FUNCTION "dos_comp_7" : VOID	// FC 9
TITLE = Dosing component 7
VERSION : 0.1
VAR_TEMP
  dosi_man : BOOL ;
END_VAR
BEGIN
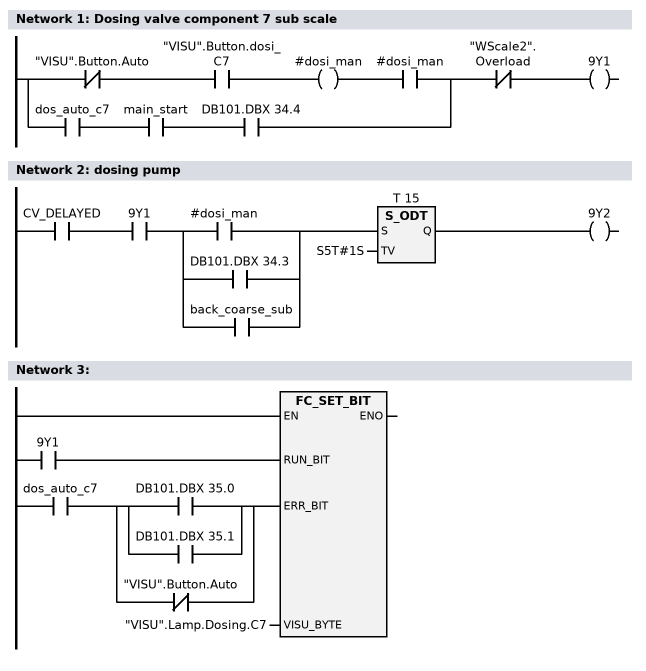
NETWORK
TITLE = Dosing valve component 7 sub scale
//automatic and manual steps
      A(;
      AN    "VISU".Button.Auto;
      A     "VISU".Button.dosi_C7;
      =     #dosi_man;
      A     #dosi_man;
      O;
      A     "dos_auto_c7";
      A     "main_start";
      A     DB101.DBX 34.4;
      );
      AN    "WScale2".Overload;
      =     "9Y1";
NETWORK
TITLE = dosing pump
//automatic and manual steps
      A     "CV_DELAYED";
      A     "9Y1";
      A(;
      O     #dosi_man;
      O     DB101.DBX 34.3;
      O     "back_coarse_sub";
      );
      L     S5T#1S;
      SD    T 15;
      NOP   0;
      NOP   0;
      NOP   0;
      A     T 15;
      =     "9Y2";
NETWORK
TITLE =
      A     "9Y1";
      =     L 1.0;
      BLD   103;
      A     "dos_auto_c7";
      A(;
      O     DB101.DBX 35.0;
      O     DB101.DBX 35.1;
      ON    "VISU".Button.Auto;
      );
      =     L 1.1;
      BLD   103;
      CALL  "FC_SET_BIT" (
           RUN_BIT                  := L 1.0,
           ERR_BIT                  := L 1.1,
           VISU_BYTE                := "VISU".Lamp.Dosing.C7);
      NOP   0;
END_FUNCTION

FUNCTION "dos_comp_8" : VOID	// FC 10
TITLE = Dosing component 8
VERSION : 0.1
VAR_TEMP
  dosi_man : BOOL ;
END_VAR
BEGIN
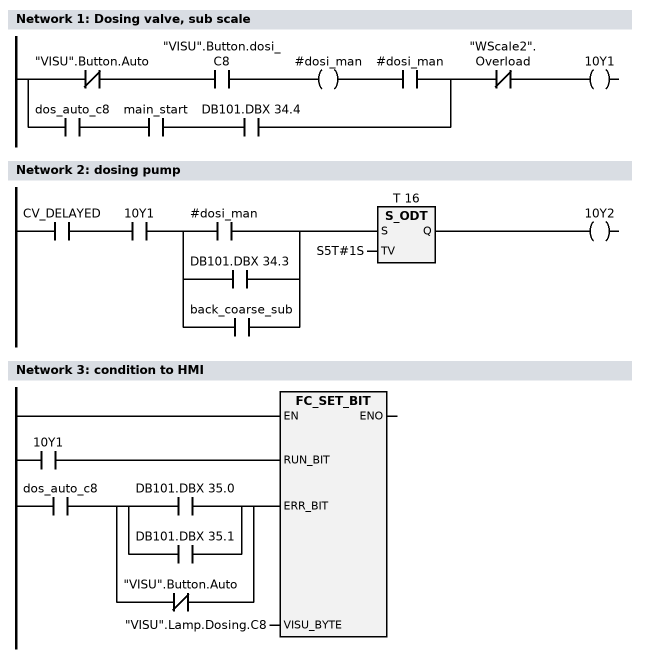
NETWORK
TITLE = Dosing valve, sub scale
//automatic and manual steps
      A(;
      AN    "VISU".Button.Auto;
      A     "VISU".Button.dosi_C8;
      =     #dosi_man;
      A     #dosi_man;
      O;
      A     "dos_auto_c8";
      A     "main_start";
      A     DB101.DBX 34.4;
      );
      AN    "WScale2".Overload;
      =     "10Y1";
NETWORK
TITLE = dosing pump
//automatic and manual steps
      A     "CV_DELAYED";
      A     "10Y1";
      A(;
      O     #dosi_man;
      O     DB101.DBX 34.3;
      O     "back_coarse_sub";
      );
      L     S5T#1S;
      SD    T 16;
      NOP   0;
      NOP   0;
      NOP   0;
      A     T 16;
      =     "10Y2";
NETWORK
TITLE = condition to HMI 
      A     "10Y1";
      =     L 1.0;
      BLD   103;
      A     "dos_auto_c8";
      A(;
      O     DB101.DBX 35.0;
      O     DB101.DBX 35.1;
      ON    "VISU".Button.Auto;
      );
      =     L 1.1;
      BLD   103;
      CALL  "FC_SET_BIT" (
           RUN_BIT                  := L 1.0,
           ERR_BIT                  := L 1.1,
           VISU_BYTE                := "VISU".Lamp.Dosing.C8);
      NOP   0;
END_FUNCTION

FUNCTION "dos_comp_9" : VOID	// FC 11
TITLE = Dosing component 9
VERSION : 0.1
VAR_TEMP
  dosi_man : BOOL ;
END_VAR
BEGIN
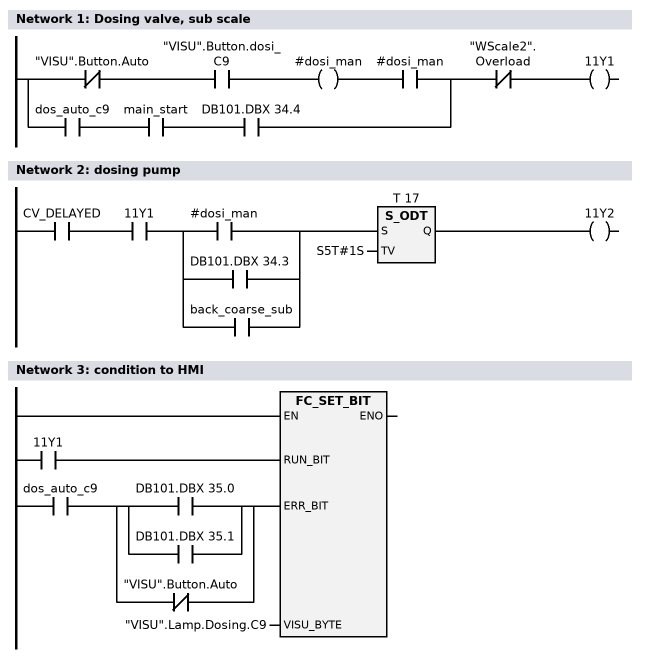
NETWORK
TITLE = Dosing valve, sub scale
//automatic and manual steps
      A(;
      AN    "VISU".Button.Auto;
      A     "VISU".Button.dosi_C9;
      =     #dosi_man;
      A     #dosi_man;
      O;
      A     "dos_auto_c9";
      A     "main_start";
      A     DB101.DBX 34.4;
      );
      AN    "WScale2".Overload;
      =     "11Y1";
NETWORK
TITLE = dosing pump
//automatic and manual steps
      A     "CV_DELAYED";
      A     "11Y1";
      A(;
      O     #dosi_man;
      O     DB101.DBX 34.3;
      O     "back_coarse_sub";
      );
      L     S5T#1S;
      SD    T 17;
      NOP   0;
      NOP   0;
      NOP   0;
      A     T 17;
      =     "11Y2";
NETWORK
TITLE = condition to HMI 
      A     "11Y1";
      =     L 1.0;
      BLD   103;
      A     "dos_auto_c9";
      A(;
      O     DB101.DBX 35.0;
      O     DB101.DBX 35.1;
      ON    "VISU".Button.Auto;
      );
      =     L 1.1;
      BLD   103;
      CALL  "FC_SET_BIT" (
           RUN_BIT                  := L 1.0,
           ERR_BIT                  := L 1.1,
           VISU_BYTE                := "VISU".Lamp.Dosing.C9);
      NOP   0;
END_FUNCTION

FUNCTION "dos_comp_10" : VOID	// FC 12
TITLE = Dosing component 10
VERSION : 0.1
VAR_TEMP
  dosi_man : BOOL ;
END_VAR
BEGIN
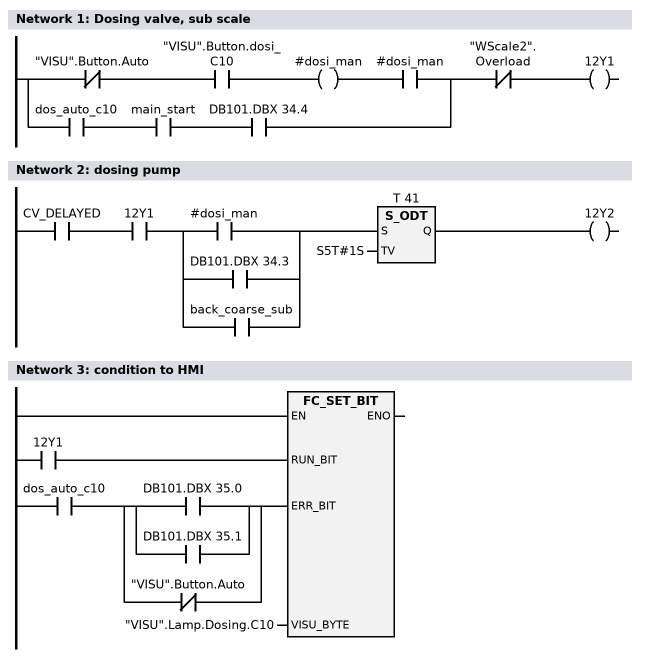
NETWORK
TITLE = Dosing valve, sub scale
//automatic and manual steps
      A(;
      AN    "VISU".Button.Auto;
      A     "VISU".Button.dosi_C10;
      =     #dosi_man;
      A     #dosi_man;
      O;
      A     "dos_auto_c10";
      A     "main_start";
      A     DB101.DBX 34.4;
      );
      AN    "WScale2".Overload;
      =     "12Y1";
NETWORK
TITLE = dosing pump
//automatic and manual steps
      A     "CV_DELAYED";
      A     "12Y1";
      A(;
      O     #dosi_man;
      O     DB101.DBX 34.3;
      O     "back_coarse_sub";
      );
      L     S5T#1S;
      SD    T 41;
      NOP   0;
      NOP   0;
      NOP   0;
      A     T 41;
      =     "12Y2";
NETWORK
TITLE = condition to HMI
      A     "12Y1";
      =     L 1.0;
      BLD   103;
      A     "dos_auto_c10";
      A(;
      O     DB101.DBX 35.0;
      O     DB101.DBX 35.1;
      ON    "VISU".Button.Auto;
      );
      =     L 1.1;
      BLD   103;
      CALL  "FC_SET_BIT" (
           RUN_BIT                  := L 1.0,
           ERR_BIT                  := L 1.1,
           VISU_BYTE                := "VISU".Lamp.Dosing.C10);
      NOP   0;
END_FUNCTION

FUNCTION "dos_comp_11" : VOID	// FC 13
TITLE = Dosing component 11
VERSION : 0.1
VAR_TEMP
  dosi_man : BOOL ;
END_VAR
BEGIN
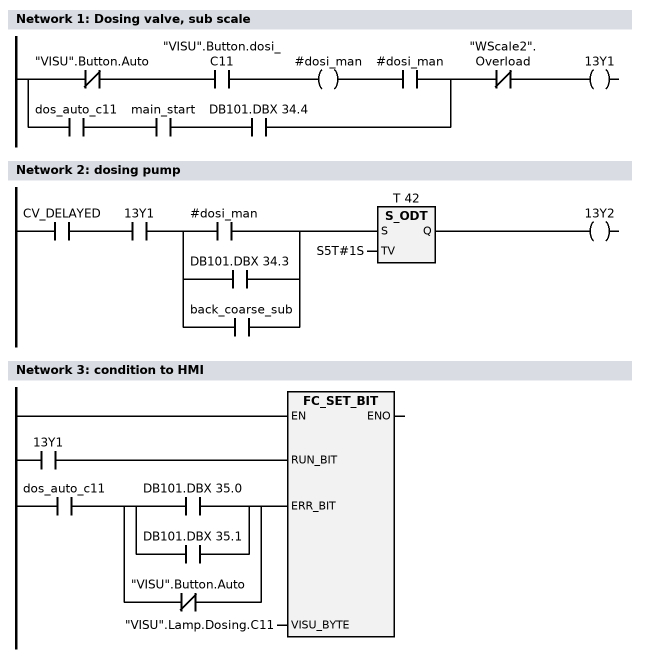
NETWORK
TITLE = Dosing valve, sub scale
//automatic and manual steps
      A(;
      AN    "VISU".Button.Auto;
      A     "VISU".Button.dosi_C11;
      =     #dosi_man;
      A     #dosi_man;
      O;
      A     "dos_auto_c11";
      A     "main_start";
      A     DB101.DBX 34.4;
      );
      AN    "WScale2".Overload;
      =     "13Y1";
NETWORK
TITLE = dosing pump
//automatic and manual steps
      A     "CV_DELAYED";
      A     "13Y1";
      A(;
      O     #dosi_man;
      O     DB101.DBX 34.3;
      O     "back_coarse_sub";
      );
      L     S5T#1S;
      SD    T 42;
      NOP   0;
      NOP   0;
      NOP   0;
      A     T 42;
      =     "13Y2";
NETWORK
TITLE = condition to HMI
      A     "13Y1";
      =     L 1.0;
      BLD   103;
      A     "dos_auto_c11";
      A(;
      O     DB101.DBX 35.0;
      O     DB101.DBX 35.1;
      ON    "VISU".Button.Auto;
      );
      =     L 1.1;
      BLD   103;
      CALL  "FC_SET_BIT" (
           RUN_BIT                  := L 1.0,
           ERR_BIT                  := L 1.1,
           VISU_BYTE                := "VISU".Lamp.Dosing.C11);
      NOP   0;
END_FUNCTION

FUNCTION "dos_comp_12" : VOID	// FC 14
TITLE = Dosing component 12
VERSION : 0.1
VAR_TEMP
  dosi_man : BOOL ;
END_VAR
BEGIN
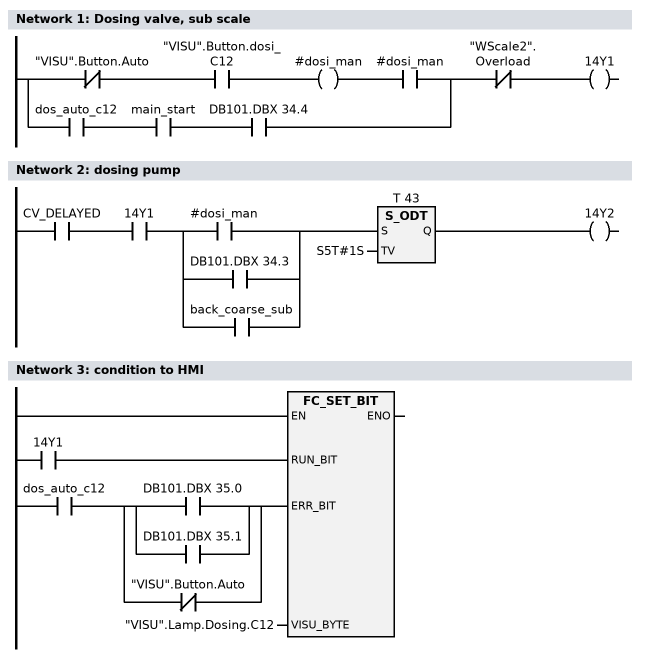
NETWORK
TITLE = Dosing valve, sub scale
//automatic and manual steps
      A(;
      AN    "VISU".Button.Auto;
      A     "VISU".Button.dosi_C12;
      =     #dosi_man;
      A     #dosi_man;
      O;
      A     "dos_auto_c12";
      A     "main_start";
      A     DB101.DBX 34.4;
      );
      AN    "WScale2".Overload;
      =     "14Y1";
NETWORK
TITLE = dosing pump
//automatic and manual steps
      A     "CV_DELAYED";
      A     "14Y1";
      A(;
      O     #dosi_man;
      O     DB101.DBX 34.3;
      O     "back_coarse_sub";
      );
      L     S5T#1S;
      SD    T 43;
      NOP   0;
      NOP   0;
      NOP   0;
      A     T 43;
      =     "14Y2";
NETWORK
TITLE = condition to HMI
      A     "14Y1";
      =     L 1.0;
      BLD   103;
      A     "dos_auto_c12";
      A(;
      O     DB101.DBX 35.0;
      O     DB101.DBX 35.1;
      ON    "VISU".Button.Auto;
      );
      =     L 1.1;
      BLD   103;
      CALL  "FC_SET_BIT" (
           RUN_BIT                  := L 1.0,
           ERR_BIT                  := L 1.1,
           VISU_BYTE                := "VISU".Lamp.Dosing.C12);
      NOP   0;
END_FUNCTION

FUNCTION "discharge_main_scale" : VOID	// FC 22
TITLE = discharge mainscale
VERSION : 0.0
VAR_TEMP
  disc_auto : BOOL ;
  disc1 : BOOL ;
  disc2 : BOOL ;
  disc3 : BOOL ;
END_VAR
BEGIN
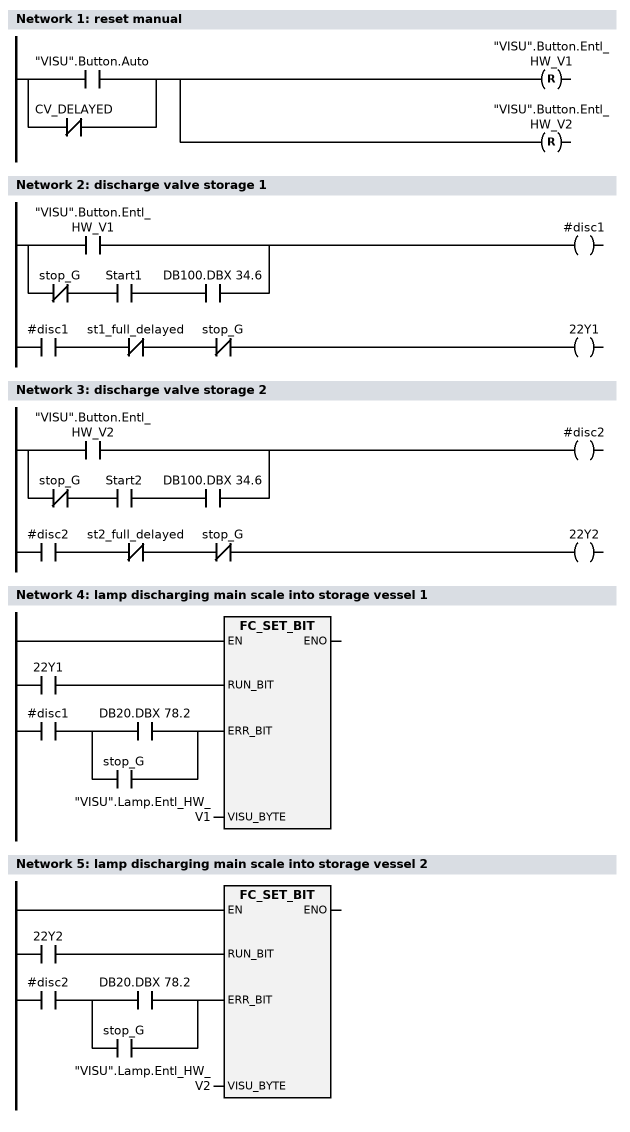
NETWORK
TITLE = reset manual
      O     "VISU".Button.Auto;
      ON    "CV_DELAYED";
      R     "VISU".Button.Entl_HW_V1;
      R     "VISU".Button.Entl_HW_V2;
NETWORK
TITLE = discharge valve storage 1
      A(;
      O     "VISU".Button.Entl_HW_V1;
      O;
      AN    "stop_G";
      A     "Start1";
      A     DB100.DBX 34.6;
      );
      =     #disc1;
      A     #disc1;
      AN    "st1_full_delayed";
      AN    "stop_G";
      =     "22Y1";
NETWORK
TITLE = discharge valve storage 2
      A(;
      O     "VISU".Button.Entl_HW_V2;
      O;
      AN    "stop_G";
      A     "Start2";
      A     DB100.DBX 34.6;
      );
      =     #disc2;
      A     #disc2;
      AN    "st2_full_delayed";
      AN    "stop_G";
      =     "22Y2";
NETWORK
TITLE = lamp discharging main scale into storage vessel 1
      A     "22Y1";
      =     L 1.0;
      BLD   103;
      A     #disc1;
      A(;
      O     DB20.DBX 78.2;
      O     "stop_G";
      );
      =     L 1.1;
      BLD   103;
      CALL  "FC_SET_BIT" (
           RUN_BIT                  := L 1.0,
           ERR_BIT                  := L 1.1,
           VISU_BYTE                := "VISU".Lamp.Entl_HW_V1);
      NOP   0;
NETWORK
TITLE = lamp discharging main scale into storage vessel 2
      A     "22Y2";
      =     L 1.0;
      BLD   103;
      A     #disc2;
      A(;
      O     DB20.DBX 78.2;
      O     "stop_G";
      );
      =     L 1.1;
      BLD   103;
      CALL  "FC_SET_BIT" (
           RUN_BIT                  := L 1.0,
           ERR_BIT                  := L 1.1,
           VISU_BYTE                := "VISU".Lamp.Entl_HW_V2);
      NOP   0;
END_FUNCTION

FUNCTION "discharge_sub_scale" : VOID	// FC 23
TITLE = discharge  sub scale
VERSION : 0.1
VAR_TEMP
  disc : BOOL ;
END_VAR
BEGIN
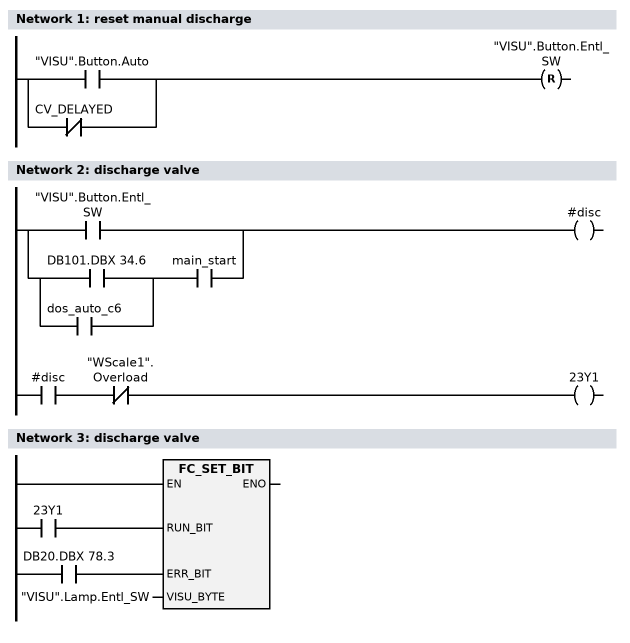
NETWORK
TITLE = reset manual discharge
      O     "VISU".Button.Auto;
      ON    "CV_DELAYED";
      R     "VISU".Button.Entl_SW;
NETWORK
TITLE = discharge valve
      A(;
      O     "VISU".Button.Entl_SW;
      O;
      A(;
      O     DB101.DBX 34.6;
      O     "dos_auto_c6";
      );
      A     "main_start";
      );
      =     #disc;
      A     #disc;
      AN    "WScale1".Overload;
      =     "23Y1";
NETWORK
TITLE = discharge valve
      A     "23Y1";
      =     L 1.0;
      BLD   103;
      A     DB20.DBX 78.3;
      =     L 1.1;
      BLD   103;
      CALL  "FC_SET_BIT" (
           RUN_BIT                  := L 1.0,
           ERR_BIT                  := L 1.1,
           VISU_BYTE                := "VISU".Lamp.Entl_SW);
      NOP   0;
END_FUNCTION

FUNCTION "agit_MS" : VOID	// FC 25
TITLE = main scale, agitator
VERSION : 0.1
BEGIN
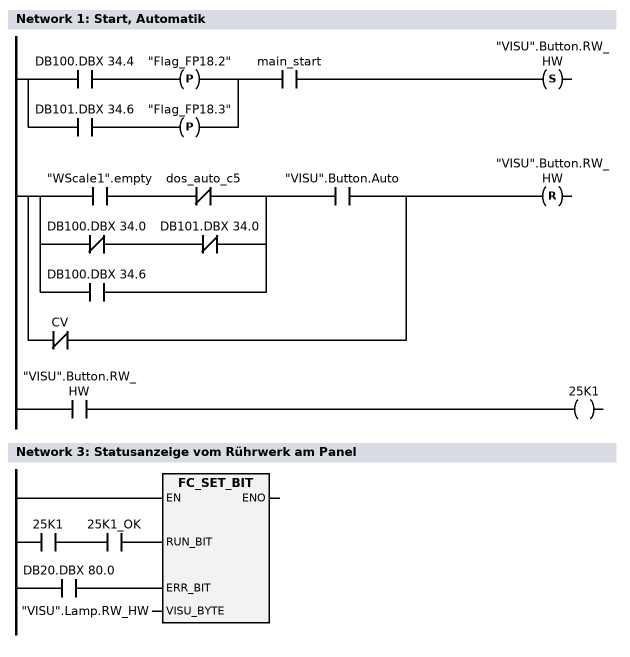
NETWORK
TITLE = Start, Automatik
      A(;
      A     DB100.DBX 34.4;
      FP    "Flag_FP18.2";
      O(;
      A     DB101.DBX 34.6;
      FP    "Flag_FP18.3";
      );
      );
      A     "main_start";
      S     "VISU".Button.RW_HW;
      A(;
      A(;
      A     "WScale1".empty;
      AN    "dos_auto_c5";
      O;
      AN    DB100.DBX 34.0;
      AN    DB101.DBX 34.0;
      O     DB100.DBX 34.6;
      );
      A     "VISU".Button.Auto;
      ON    "CV";
      );
      R     "VISU".Button.RW_HW;
      A     "VISU".Button.RW_HW;
      =     "25K1";
NETWORK
TITLE = Schütz auf Rückmeldung prüfen
      A(;
      X     "25K1";
      X     "25K1_OK";
      );
      A     "CV_DELAYED";
      L     S5T#1S;
      SD    T 18;
      NOP   0;
      NOP   0;
      NOP   0;
      A     T 18;
      =     DB20.DBX 80.0;
NETWORK
TITLE = Statusanzeige vom Rührwerk am Panel
      A     "25K1";
      A     "25K1_OK";
      =     L 0.0;
      BLD   103;
      A     DB20.DBX 80.0;
      =     L 0.1;
      BLD   103;
      CALL  "FC_SET_BIT" (
           RUN_BIT                  := L 0.0,
           ERR_BIT                  := L 0.1,
           VISU_BYTE                := "VISU".Lamp.RW_HW);
      NOP   0;
END_FUNCTION

FUNCTION "aigt_level_storage1" : VOID	// FC 26
TITLE = agit_level storage vessel 1
VERSION : 0.1
VAR_TEMP
  imp : BOOL ;
END_VAR
BEGIN
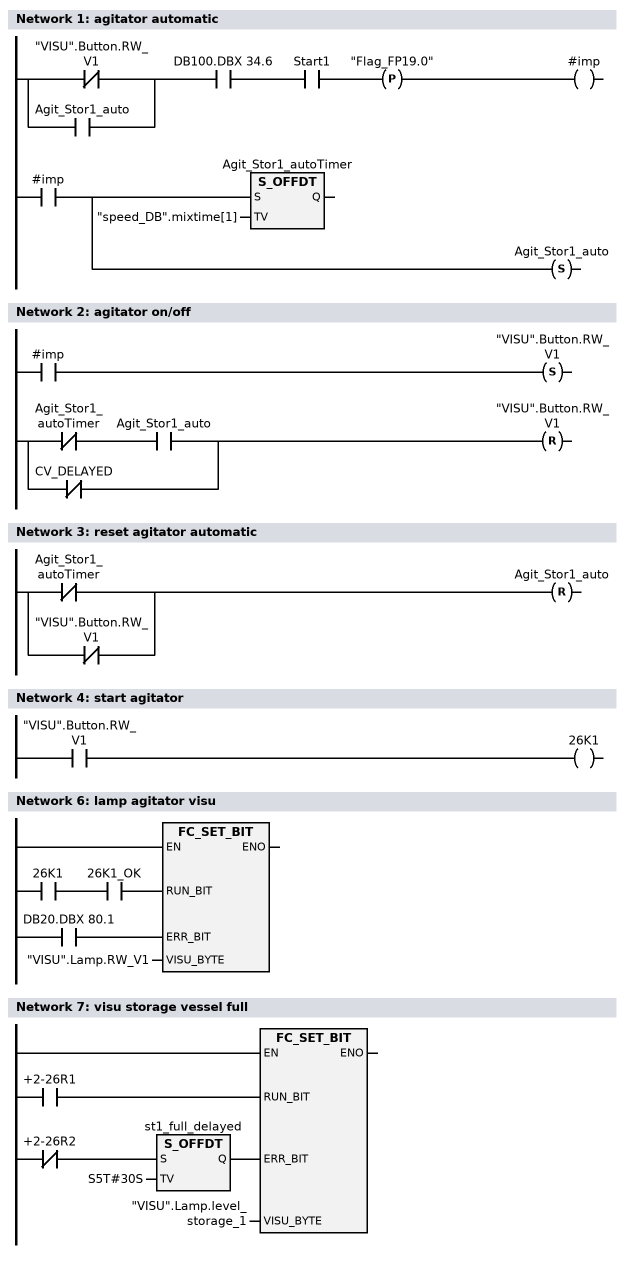
NETWORK
TITLE = agitator automatic
      A(;
      ON    "VISU".Button.RW_V1;
      O     "Agit_Stor1_auto";
      );
      A     DB100.DBX 34.6;
      A     "Start1";
      FP    "Flag_FP19.0";
      =     #imp;
      A     #imp;
      =     L 1.0;
      A     L 1.0;
      L     "speed_DB".mixtime[1];
      SF    "Agit_Stor1_autoTimer";
      NOP   0;
      NOP   0;
      NOP   0;
      NOP   0;
      A     L 1.0;
      BLD   102;
      S     "Agit_Stor1_auto";
NETWORK
TITLE = agitator on/off
      A     #imp;
      S     "VISU".Button.RW_V1;
      A(;
      AN    "Agit_Stor1_autoTimer";
      A     "Agit_Stor1_auto";
      ON    "CV_DELAYED";
      );
      R     "VISU".Button.RW_V1;
      NOP   0;
NETWORK
TITLE = reset agitator automatic
      ON    "Agit_Stor1_autoTimer";
      ON    "VISU".Button.RW_V1;
      R     "Agit_Stor1_auto";
NETWORK
TITLE = start agitator
      A     "VISU".Button.RW_V1;
      =     "26K1";
NETWORK
TITLE = fault contactor/circuit breaker
      A(;
      X     "26K1";
      X     "26K1_OK";
      );
      A     "CV_DELAYED";
      L     S5T#1S;
      SD    T 10;
      NOP   0;
      NOP   0;
      NOP   0;
      A     T 10;
      =     DB20.DBX 80.1;
NETWORK
TITLE = lamp agitator visu
      A     "26K1";
      A     "26K1_OK";
      =     L 1.0;
      BLD   103;
      A     DB20.DBX 80.1;
      =     L 1.1;
      BLD   103;
      CALL  "FC_SET_BIT" (
           RUN_BIT                  := L 1.0,
           ERR_BIT                  := L 1.1,
           VISU_BYTE                := "VISU".Lamp.RW_V1);
      NOP   0;
NETWORK
TITLE = visu storage vessel full
      A     "+2-26R1";
      =     L 1.0;
      BLD   103;
      A(;
      AN    "+2-26R2";
      L     S5T#30S;
      SF    "st1_full_delayed";
      NOP   0;
      NOP   0;
      NOP   0;
      A     "st1_full_delayed";
      );
      =     L 1.1;
      BLD   103;
      CALL  "FC_SET_BIT" (
           RUN_BIT                  := L 1.0,
           ERR_BIT                  := L 1.1,
           VISU_BYTE                := "VISU".Lamp.level_storage_1);
      NOP   0;
END_FUNCTION

FUNCTION "aigt_level_storage2" : VOID	// FC 27
TITLE = agit_level storage vessel 2
VERSION : 0.1
VAR_TEMP
  imp : BOOL ;
END_VAR
BEGIN
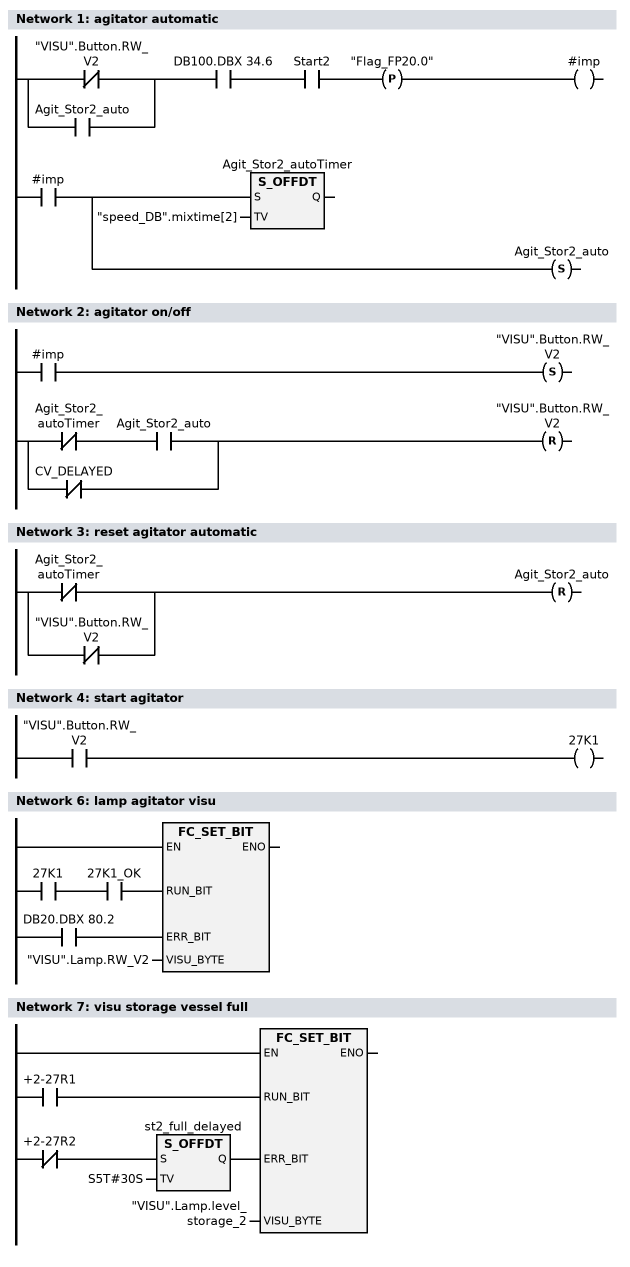
NETWORK
TITLE = agitator automatic
      A(;
      ON    "VISU".Button.RW_V2;
      O     "Agit_Stor2_auto";
      );
      A     DB100.DBX 34.6;
      A     "Start2";
      FP    "Flag_FP20.0";
      =     #imp;
      A     #imp;
      =     L 1.0;
      A     L 1.0;
      L     "speed_DB".mixtime[2];
      SF    "Agit_Stor2_autoTimer";
      NOP   0;
      NOP   0;
      NOP   0;
      NOP   0;
      A     L 1.0;
      BLD   102;
      S     "Agit_Stor2_auto";
NETWORK
TITLE = agitator on/off
      A     #imp;
      S     "VISU".Button.RW_V2;
      A(;
      AN    "Agit_Stor2_autoTimer";
      A     "Agit_Stor2_auto";
      ON    "CV_DELAYED";
      );
      R     "VISU".Button.RW_V2;
      NOP   0;
NETWORK
TITLE = reset agitator automatic
      ON    "Agit_Stor2_autoTimer";
      ON    "VISU".Button.RW_V2;
      R     "Agit_Stor2_auto";
NETWORK
TITLE = start agitator
      A     "VISU".Button.RW_V2;
      =     "27K1";
NETWORK
TITLE = fault contactor/circuit breaker
      A(;
      X     "27K1";
      X     "27K1_OK";
      );
      A     "CV_DELAYED";
      L     S5T#1S;
      SD    T 22;
      NOP   0;
      NOP   0;
      NOP   0;
      A     T 22;
      =     DB20.DBX 80.2;
NETWORK
TITLE = lamp agitator visu
      A     "27K1";
      A     "27K1_OK";
      =     L 1.0;
      BLD   103;
      A     DB20.DBX 80.2;
      =     L 1.1;
      BLD   103;
      CALL  "FC_SET_BIT" (
           RUN_BIT                  := L 1.0,
           ERR_BIT                  := L 1.1,
           VISU_BYTE                := "VISU".Lamp.RW_V2);
      NOP   0;
NETWORK
TITLE = visu storage vessel full
      A     "+2-27R1";
      =     L 1.0;
      BLD   103;
      A(;
      AN    "+2-27R2";
      L     S5T#30S;
      SF    "st2_full_delayed";
      NOP   0;
      NOP   0;
      NOP   0;
      A     "st2_full_delayed";
      );
      =     L 1.1;
      BLD   103;
      CALL  "FC_SET_BIT" (
           RUN_BIT                  := L 1.0,
           ERR_BIT                  := L 1.1,
           VISU_BYTE                := "VISU".Lamp.level_storage_2);
      NOP   0;
END_FUNCTION

FUNCTION "filling_vat" : VOID	// FC 29
TITLE = Vat VITS filling out from storage 1
VERSION : 0.1
VAR_TEMP
  valve_1 : BOOL ;
  valve_2 : BOOL ;
END_VAR
BEGIN
NETWORK
TITLE = Filling ON/OFF
//"VISU".Button.filling_1
      A(;
      A(;
      A     "VISU".Button.filling_1;
      AN    "+4-29R1";
      S     "VITS1_FILLING_ON/OFF";
      A(;
      ON    "VISU".Button.filling_1;
      ON    "+4-29R2";
      );
      R     "VITS1_FILLING_ON/OFF";
      A     "VITS1_FILLING_ON/OFF";
      );
      AN    DB20.DBX 83.0;
      O(;
      A     "VISU".Button.fillvalve_1;
      L     S5T#3S;
      SD    "VITS1_TIPP_TIMER";
      A     "VISU".Button.filling_3;
      R     "VITS1_TIPP_TIMER";
      NOP   0;
      NOP   0;
      A     "VITS1_TIPP_TIMER";
      );
      );
      =     #valve_1;
      A     #valve_1;
      A     "+VTITS-K1";
      L     S5T#1S;
      SF    T 44;
      NOP   0;
      NOP   0;
      NOP   0;
      A     T 44;
      =     "+4-29Y1";
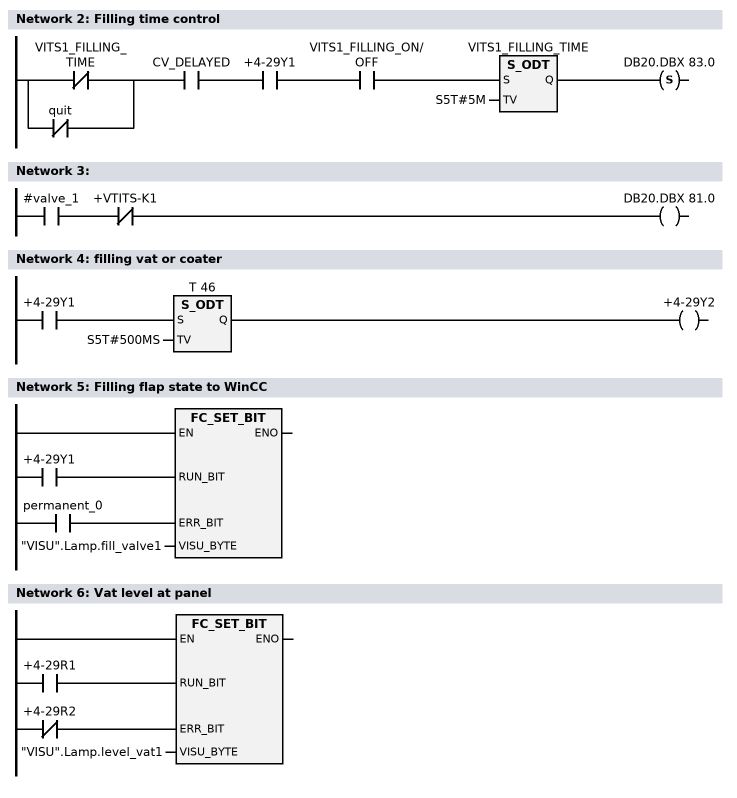
NETWORK
TITLE = Filling time control
      A(;
      ON    "VITS1_FILLING_TIME";
      ON    "quit";
      );
      A     "CV_DELAYED";
      A     "+4-29Y1";
      A     "VITS1_FILLING_ON/OFF";
      L     S5T#5M;
      SD    "VITS1_FILLING_TIME";
      NOP   0;
      NOP   0;
      NOP   0;
      A     "VITS1_FILLING_TIME";
      S     DB20.DBX 83.0;
NETWORK
TITLE =
      A     #valve_1;
      AN    "+VTITS-K1";
      =     DB20.DBX 81.0;
NETWORK
TITLE = filling vat or coater
      A     "+4-29Y1";
      L     S5T#500MS;
      SD    T 46;
      NOP   0;
      NOP   0;
      NOP   0;
      A     T 46;
      =     "+4-29Y2";
NETWORK
TITLE = Filling flap state to WinCC
      A     "+4-29Y1";
      =     L 1.0;
      BLD   103;
      A     "permanent_0";
      =     L 1.1;
      BLD   103;
      CALL  "FC_SET_BIT" (
           RUN_BIT                  := L 1.0,
           ERR_BIT                  := L 1.1,
           VISU_BYTE                := "VISU".Lamp.fill_valve1);
      NOP   0;
NETWORK
TITLE = Vat level at panel
      A     "+4-29R1";
      =     L 1.0;
      BLD   103;
      AN    "+4-29R2";
      =     L 1.1;
      BLD   103;
      CALL  "FC_SET_BIT" (
           RUN_BIT                  := L 1.0,
           ERR_BIT                  := L 1.1,
           VISU_BYTE                := "VISU".Lamp.level_vat1);
      NOP   0;
END_FUNCTION

FUNCTION "filling_coater" : VOID	// FC 30
TITLE = Coater VITS
VERSION : 0.1
BEGIN
NETWORK
TITLE = Filling ON/OFF
//"VISU".Button.filling_2
      A(;
      A     "VISU".Button.filling_2;
      AN    "+4-30R1";
      S     "VITS2_FILLING_ON/OFF";
      A(;
      ON    "VISU".Button.filling_2;
      ON    "+4-30R2";
      );
      R     "VITS2_FILLING_ON/OFF";
      A     "VITS2_FILLING_ON/OFF";
      );
      AN    DB20.DBX 83.1;
      O(;
      A     "VISU".Button.fillvalve_2;
      L     S5T#3S;
      SD    "VITS2_TIPP_TIMER";
      NOP   0;
      NOP   0;
      NOP   0;
      A     "VITS2_TIPP_TIMER";
      );
      =     "+4-30Y1";
      =     "+4-30Y2";
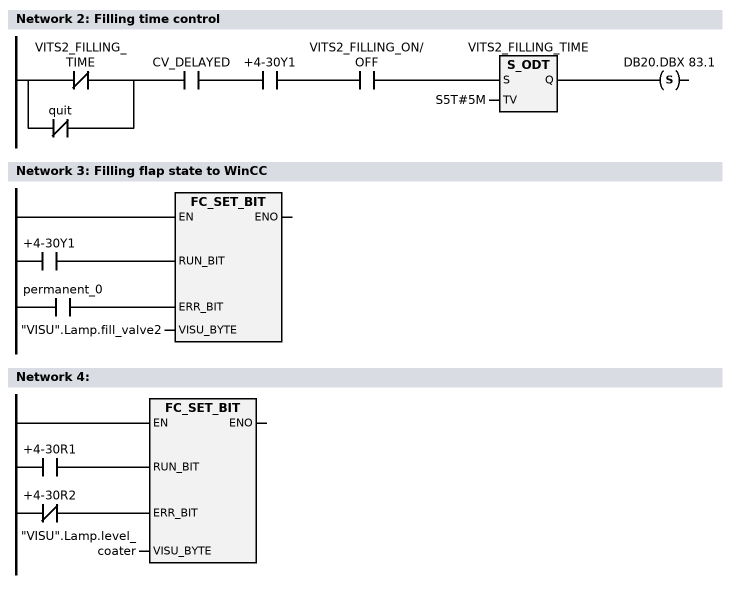
NETWORK
TITLE = Filling time control
      A(;
      ON    "VITS2_FILLING_TIME";
      ON    "quit";
      );
      A     "CV_DELAYED";
      A     "+4-30Y1";
      A     "VITS2_FILLING_ON/OFF";
      L     S5T#5M;
      SD    "VITS2_FILLING_TIME";
      NOP   0;
      NOP   0;
      NOP   0;
      A     "VITS2_FILLING_TIME";
      S     DB20.DBX 83.1;
NETWORK
TITLE = Filling flap state to WinCC
      A     "+4-30Y1";
      =     L 0.0;
      BLD   103;
      A     "permanent_0";
      =     L 0.1;
      BLD   103;
      CALL  "FC_SET_BIT" (
           RUN_BIT                  := L 0.0,
           ERR_BIT                  := L 0.1,
           VISU_BYTE                := "VISU".Lamp.fill_valve2);
      NOP   0;
NETWORK
TITLE =
      A     "+4-30R1";
      =     L 0.0;
      BLD   103;
      AN    "+4-30R2";
      =     L 0.1;
      BLD   103;
      CALL  "FC_SET_BIT" (
           RUN_BIT                  := L 0.0,
           ERR_BIT                  := L 0.1,
           VISU_BYTE                := "VISU".Lamp.level_coater);
      NOP   0;
END_FUNCTION

FUNCTION "coater circ" : VOID	// FC 31
TITLE = Coater circulation
VERSION : 0.1
VAR_TEMP
  fill_time : S5TIME ;
  fill_vat : BOOL ;
END_VAR
BEGIN
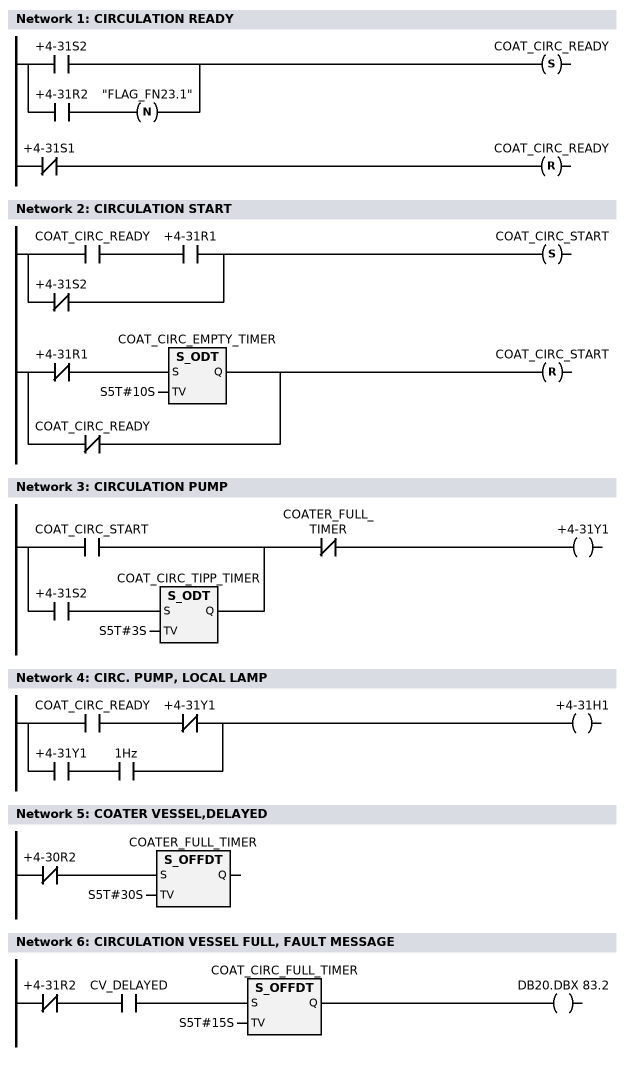
NETWORK
TITLE = CIRCULATION READY
      A(;
      O     "+4-31S2";
      O(;
      A     "+4-31R2";
      FN    "FLAG_FN23.1";
      );
      );
      S     "COAT_CIRC_READY";
      AN    "+4-31S1";
      R     "COAT_CIRC_READY";
      NOP   0;
NETWORK
TITLE = CIRCULATION START
      A(;
      A     "COAT_CIRC_READY";
      A     "+4-31R1";
      ON    "+4-31S2";
      );
      S     "COAT_CIRC_START";
      A(;
      O(;
      AN    "+4-31R1";
      L     S5T#10S;
      SD    "COAT_CIRC_EMPTY_TIMER";
      NOP   0;
      NOP   0;
      NOP   0;
      A     "COAT_CIRC_EMPTY_TIMER";
      );
      ON    "COAT_CIRC_READY";
      );
      R     "COAT_CIRC_START";
      NOP   0;
NETWORK
TITLE = CIRCULATION PUMP
      A(;
      O     "COAT_CIRC_START";
      O(;
      A     "+4-31S2";
      L     S5T#3S;
      SD    "COAT_CIRC_TIPP_TIMER";
      NOP   0;
      NOP   0;
      NOP   0;
      A     "COAT_CIRC_TIPP_TIMER";
      );
      );
      AN    "COATER_FULL_TIMER";
      =     "+4-31Y1";
NETWORK
TITLE = CIRC. PUMP, LOCAL LAMP
      A     "COAT_CIRC_READY";
      AN    "+4-31Y1";
      O;
      A     "+4-31Y1";
      A     "1Hz";
      =     "+4-31H1";
NETWORK
TITLE = COATER VESSEL,DELAYED
      AN    "+4-30R2";
      L     S5T#30S;
      SF    "COATER_FULL_TIMER";
      NOP   0;
      NOP   0;
      NOP   0;
      NOP   0;
NETWORK
TITLE = CIRCULATION VESSEL FULL, FAULT MESSAGE
      AN    "+4-31R2";
      A     "CV_DELAYED";
      L     S5T#15S;
      SF    "COAT_CIRC_FULL_TIMER";
      NOP   0;
      NOP   0;
      NOP   0;
      A     "COAT_CIRC_FULL_TIMER";
      =     DB20.DBX 83.2;
END_FUNCTION

FUNCTION "control_FC" : VOID	// FC 60
TITLE = Control FC
VERSION : 0.1
VAR_TEMP
  t_busy : BOOL ;
END_VAR
BEGIN
NETWORK
TITLE = manual operating
      CALL  "del_ins_line";
      CALL  "Transfer_Recipe";
      CALL  "Rec_handling";
NETWORK
TITLE = zero Gravimet
      L     DB21.DBB 8;	// rem Starts
      L     0;
      <>I;
      AN    "Auto_DB".automatic;
      S     "zero";
      CALL  "zero_FC";
NETWORK
TITLE = scale signals
      A     "cancel_G";
      =     DB100.DBX 34.5;
      =     DB101.DBX 34.5;
      A     "stop_G";
      A     "main_start";
      A     DB100.DBX 34.2;
      =     DB100.DBX 35.5;
      A     "stop_G";
      A     "main_start";
      A     DB101.DBX 34.2;
      =     DB101.DBX 35.5;
      A     "quit";
      R     DB100.DBX 35.2;
      R     DB101.DBX 35.2;
NETWORK
TITLE = Cascading
      L     "Cascad_DW";
      RLD   1;
      T     "Cascad_DW";
NETWORK
TITLE = main scale
      CALL  "SiwarexCS" , "WScale1" (
           ADRESSE                  := 272,
           ABZUGSWAAGE              := FALSE,
           KAS_SIWAREX              := TRUE,
           CPU_Start_Bit            := "CPU_Restart",
           ANLAUFTIMER              := "StartupTimer",
           Quitt                    := "quit",
           StillTimer               := T 100,
           EmptyTimer               := T 101,
           DosiControlTimer         := T 102,
           StepTimer                := T 103);
      CALL  "Dosing" , "DScale1" (
           scale_nr                 := 1,
           Work_DB                  := 26,
           Weigh_DB                 := 10,
           mix_timer                := T 104,
           step_scale1              := "Auto_DB".Step_scale1,
           step_scale2              := "Auto_DB".Step_scale2,
           step_scale3              := "init_DB".max_step,
           step_scale4              := "init_DB".max_step,
           Dosi_Bits                := "Dosibits");
NETWORK
TITLE = Timers
      L     T 101;
      A     "WScale1".discharge;
      JC    M001;
      L     T 103;
      A     "WScale1".StepTime;
      JC    M001;
      L     T 104;
      A     DB100.DBX 35.4;
      JC    M001;
      L     0;
M001: L     60;
      /I;
      T     "HMI_DB".Scale1_timers;
NETWORK
TITLE = fault messages
      A     DB100.DBX 35.0;
      S     DB20.DBX 73.1;
      A     DB100.DBX 35.1;
      AN    DB100.DBX 35.5;
      S     DB20.DBX 73.2;
      A     DB100.DBX 35.5;
      S     DB20.DBX 73.3;
NETWORK
TITLE = sub scale
      CALL  "SiwarexCS" , "WScale2" (
           ADRESSE                  := 280,
           ABZUGSWAAGE              := FALSE,
           KAS_SIWAREX              := TRUE,
           CPU_Start_Bit            := "CPU_Restart",
           ANLAUFTIMER              := "StartupTimer",
           Quitt                    := "quit",
           StillTimer               := T 105,
           EmptyTimer               := T 106,
           DosiControlTimer         := T 107,
           StepTimer                := T 108);
      CALL  "Dosing" , "DScale2" (
           scale_nr                 := 2,
           Work_DB                  := 26,
           Weigh_DB                 := 11,
           mix_timer                := T 109,
           step_scale1              := "Auto_DB".Step_scale1,
           step_scale2              := "Auto_DB".Step_scale2,
           step_scale3              := "init_DB".max_step,
           step_scale4              := "init_DB".max_step,
           Dosi_Bits                := "Dosibits");
NETWORK
TITLE = Timers
      L     T 106;
      A     "WScale2".discharge;
      JC    M002;
      L     T 108;
      A     "WScale2".StepTime;
      JC    M002;
      L     T 109;
      A     DB101.DBX 35.4;
      JC    M002;
      L     0;
M002: L     60;
      /I;
      T     "HMI_DB".Scale2_timers;
NETWORK
TITLE = fault messages sub scale
      A     DB101.DBX 35.0;
      S     DB20.DBX 72.1;
      A     DB101.DBX 35.1;
      AN    DB101.DBX 35.5;
      S     DB20.DBX 72.2;
      A     DB101.DBX 35.5;
      S     DB20.DBX 72.3;
NETWORK
TITLE = rated value total main scale while discharging sub scale
      A     DB101.DBX 34.6;
      FP    "Flag_FP211.0";
      JCN   M003;
      L     DB101.DBD 44;
      L     DB100.DBD 44;
      +R;
      T     DB100.DBD 44;
      L     0;
      T     DB100.DBD 22;
M003: NOP   0;
NETWORK
TITLE = clear starts Gravimet
      AN    "zero";
      AN    DB100.DBX 34.0;
      AN    DB101.DBX 34.0;
      R     "Auto_DB".automatic;
      S     "del_starts_G";
END_FUNCTION

FUNCTION "zero_FC" : VOID	// FC 61
TITLE = Waage nullen
//know_how_protect
//
VERSION : 0.0
VAR_TEMP
  loop_ctr1 : INT ;
  loop_ctr2 : INT ;
  Sum_comp : INT ;
  comp_nr : INT ;
  action : INT ;
  scale_nr : INT ;
  DB_ptr : INT ;
  percent : REAL ;
  Sum_main : REAL ;
  Sum_Sub : REAL ;
  Sum_Col : REAL ;
  Rated_val : REAL ;
  Sum_ptr : DINT ;
  Col_flag : BOOL ;
  Temp_err : BOOL ;
  ptr1 : DINT ;
  ptr2 : DINT ;
  recipe : INT ;
  agit_time : INT ;
  Work_DB : INT ;
  CP_DB : INT ;
  Rec_DB : INT ;
  db_write_CP_date : WORD ;
END_VAR
BEGIN
NETWORK
TITLE = Startnummer bestimmen
      AN    "zero";
      BEC;
      L     0;
      A     "Auto_DB".rem_start1;
      JC    M001;
      L     1;
      A     "Auto_DB".rem_start2;
      JC    M001;
      L     2;
M001: T     "Auto_DB".Start_G;
NETWORK
TITLE = Prozentzahl und RezNr für Start
      L     "Auto_DB".Start_G;
      L     30;	// 15 Datenworte pro Start
      *D;
      SLD   3;	// 3 wg Ptr
      LAR1;
      OPN   "Start_DB";
      L     0;
      L     DBW [AR1,P#0.0];
      ==I;
      S     DB20.DBX 76.7;
      JC    M002;	// Rezeptnr 0
      T     #recipe;
      OPN   "Start_DB";
      L     0;
      L     DBW [AR1,P#2.0];
      ==I;
      S     DB20.DBX 76.0;
      JC    M002;	// keine Prozentzahl eingegeben
      ITD;
      DTR;
      L     1.000000e+02;
      /R;
      T     #percent;
NETWORK
TITLE = waiting for zero and standstill
      A     "zero_wait";
      JC    M004;
      AN    "WScale1".Standstill;
      BEC;
      AN    "WScale2".Standstill;
      BEC;
NETWORK
TITLE = zero point check, sub- and mainscale
      A     "WScale1".no_zero;
      S     DB20.DBX 73.0;
      S     "WScale1".show_zero;
      A     "WScale2".no_zero;
      S     DB20.DBX 72.0;
      S     "WScale2".show_zero;
      O     "WScale1".no_zero;
      O     "WScale2".no_zero;
      JC    M002;	// Nullfehler  
NETWORK
TITLE = nullen
      L     1;
      T     DB100.DBW 42;
      T     DB101.DBW 42;
      L     3;
      T     "WScale1".Command;
      S     "WScale1".WriteCommand;
      T     "WScale2".Command;
      S     "WScale2".WriteCommand;
      A     "permanent_1";
      S     "zero_wait";
M004: O     "WScale1".WriteCommand;
      O     "WScale2".WriteCommand;
      A     "zero_wait";
      BEC;
      R     "zero_wait";
NETWORK
TITLE = DB-Number set
      L     26;
      T     #Work_DB;
      L     "Auto_DB".Start_G;
      L     150;
      +I;
      T     #Rec_DB;
NETWORK
TITLE = Work-DB reset
      LAR1  P#0.0;
      L     "init_DB".max_step;
      L     "init_DB".step_size;
      *I;
      L     2;	// Word
      /I;
      OPN   DB [#Work_DB];
M006: T     #loop_ctr2;
      L     0;
      T     DBW [AR1,P#0.0];
      +AR1  P#2.0;
      L     #loop_ctr2;
      LOOP  M006;
NETWORK
TITLE = end, if transfer is active
      L     "Recipe_transfer_byte";
      L     0;
      <>I;
      BEC;
NETWORK
TITLE =
      L     0;
      T     #Sum_main;
      T     #Sum_Sub;	// 5 Words pro Komponente
      T     #Sum_Col;	// 15Words CP Kopf
      T     #Sum_comp;
      T     #loop_ctr1;
      LAR1;
      L     "init_DB".max_step;
      R     #Col_flag;
M015: T     #loop_ctr1;
      OPN   DB [#Rec_DB];
      L     0;
      L     DBW [AR1,P#0.0];
      T     #action;
      ==I;
      JC    M013;
      L     DBW [AR1,P#4.0];
      T     #agit_time;
      L     #action;
      L     W#16#FF;
      AW;
      L     1;
      >I;
      JC    M014;
      L     0;
      L     DBW [AR1,P#2.0];
      T     #comp_nr;
      ==I;
      JC    M013;
      L     0.000000e+00;
      L     DBD [AR1,P#6.0];
      T     #Rated_val;
      CALL  "comp_scale" (
           component                := #comp_nr,
           scale_nr                 := #scale_nr);
      L     #scale_nr;
      L     B#16#FF;
      <>I;
      JC    nosp;
      L     1;
      T     #scale_nr;
nosp: L     0;
      L     #scale_nr;
      ==I;
      S     DB20.DBX 76.1;	// Komponente ungültig
      JC    M002;
      L     #scale_nr;
      L     3;
      ==I;
      S     #Col_flag;
      L     #scale_nr;
      L     3;
      >I;
      S     DB20.DBX 76.1;	// Komponente ungültig
      JC    M002;
      L     #comp_nr;
      L     #Sum_comp;
      +I;
      T     #Sum_comp;
      L     #scale_nr;
      L     9;
      +I;
      T     #DB_ptr;
      OPN   DB [#DB_ptr];
      L     DBD 100;
      L     #Rated_val;
      <R;
      S     DB20.DBX 76.2;	//Sollwert > Wägebereich
      JC    M002;
      L     #scale_nr;
      DEC   1;
      L     4;
      *D;
      SLD   3;
      L     P#18.0;
      +D;
      T     #Sum_ptr;
      L     #Rated_val;
      L     LD [#Sum_ptr];
      +R;
      T     LD [#Sum_ptr];
      L     #percent;
      L     #Rated_val;
      *R;
M014: OPN   DB [#Work_DB];
      T     DBD [AR1,P#6.0];
      L     #action;
      T     DBW [AR1,P#0.0];
      L     #comp_nr;
      T     DBW [AR1,P#2.0];
      L     #agit_time;
      T     DBW [AR1,P#4.0];
M013: L     "init_DB".step_size;
      SLD   3;
      +AR1;
      L     #loop_ctr1;
      LOOP  M015;
NETWORK
TITLE = Startwert initialisieren
      L     0;
      L     #Sum_comp;
      ==I;
      S     DB20.DBX 76.3;	//Keine Komponente
      JC    M002;
      L     #Sum_main;
      L     #Sum_Sub;
      +R;
      T     #Sum_main;
      L     0.000000e+00;
      ==R;
      A(;
      L     #Sum_Col;
      ==R;
      );
      S     DB20.DBX 76.4;	//Keine Sollwerte eingegeben
      JC    M002;
      L     #Sum_main;
      L     "WScale1".SP.Range;
      >R;
      S     DB20.DBX 76.5;	// Summe der Sollwerte > 
      JC    M002;
      AN    #Col_flag;
      JC    M007;
      L     #Sum_Col;
      L     DB12.DBD 100;
      >R;
      S     DB20.DBX 76.6;
      JC    M002;
      OPN   "init_DB";
      L     P#3.0;
      T     #ptr1;
      L     P#6.0;
      T     #ptr2;
      L     4;
M008: T     #loop_ctr1;
      A     M [#ptr1];
      A     DBX [#ptr2];
      JC    M007;
      L     #ptr1;
      L     1;
      +D;
      T     #ptr1;
      L     #ptr2;
      L     1;
      +D;
      T     #ptr2;
      L     #loop_ctr1;
      LOOP  M008;
      S     DB20.DBX 73.6;	//nix Farbwaage nach Papis Art möglich
      JU    M002;
M007: NOP   0;
NETWORK
TITLE =
// (network holds code this reader does not know; not shown)
NETWORK
TITLE =  Chargenprotokoll löschen
      LAR1  P#0.0;
      L     "init_DB".max_step;
      L     5;	// 5 Words pro Komponente
      *I;
      L     15;	// 15 Words CPKopf
      +I;
      OPN   DB [#CP_DB];
M012: T     #loop_ctr1;
      L     0;
      T     DBW [AR1,P#0.0];
      +AR1  P#2.0;
      L     #loop_ctr1;
      LOOP  M012;
NETWORK
TITLE = Startwerte initialisieren
// Rezept in CP
      CALL  "DB_Transfer" (
           SOURCE_DB                := 2,
           SOURCE_BYTE              := L#8,
           DRAIN_DB                 := #CP_DB,
           DRAIN_BYTE               := L#8,
           LENGTH                   := 8,
           R_VAL                    := "HMI_DB".blk_ret_val);
      OPN   DB [#CP_DB];
      L     #recipe;
      T     DBW 0;
      L     "Auto_DB".Start_G;
      L     30;
      *D;
      SLD   3;
      LAR1;
      OPN   "Start_DB";
      L     DBD [AR1,P#4.0];
      L     1;
      +D;
      T     DBD [AR1,P#4.0];
      OPN   DB [#CP_DB];
      T     DBD 2;
      L     "Auto_DB".Start_G;
      INC   1;
      OPN   DB [#CP_DB];
      T     DBW 6;
      A     "zero";
      S     "Auto_DB".automatic;
      R     "zero";
      S     DB100.DBX 34.0;
      S     DB100.DBX 34.1;
      L     0;
      T     "Auto_DB".Step_scale1;
      S     DB101.DBX 34.0;
      S     DB101.DBX 34.1;
      L     0;
      T     "Auto_DB".Step_scale2;
      BEU;
NETWORK
TITLE =
M002: S     "del_starts_G";
      R     "zero";
      R     "main_start";
END_FUNCTION

FUNCTION "BatchReport" : VOID	// FC 65
VERSION : 0.0
VAR_INPUT
  start_nr : BYTE ;
  scale_nr : INT ;
  step : INT ;
  comp : INT ;
  rated_val : REAL ;
  real_val : REAL ;
END_VAR
VAR_TEMP
  DBpointer : WORD ;
  CP_DB : WORD ;
END_VAR
BEGIN
NETWORK
TITLE =
      L     "HMI_DB".CP_DB_WRITE;	// CP for Gravimet
      T     #CP_DB;
NETWORK
TITLE =
      L     #step;
      DEC   1;
      L     P#10.0;	// Größe eines CP-feldes
      *D;
      L     P#30.0;	// Header
      +D;
      LAR1;
      OPN   DB [#CP_DB];	//DB-Zeiger
      L     #comp;	//Komp. Nummer
      T     DBW [AR1,P#0.0];
      L     30;
      +I;
      T     #DBpointer;
      L     #rated_val;
      T     DBD [AR1,P#2.0];
      L     #real_val;
      T     DBD [AR1,P#6.0];
      L     #start_nr;	//(0-n; 0=Start1)
      L     30;
      *D;
      SLD   3;
      LAR1;
      OPN   "Start_DB";
      L     #real_val;
      L     DBD [AR1,P#8.0];
      +R;
      T     DBD [AR1,P#8.0];
      OPN   DB [#DBpointer];
      L     DBD 0;	// Tankinhalt
      L     #real_val;	//  minus Istwert
      -R;
      JP    tpos;	// positiv?
      L     0;	// nein dann Tankinhalt =0
tpos: OPN   DB [#DBpointer];
      T     DBD 0;
      L     DBD 4;	// Verbrauch
      L     #real_val;	// + Istwert
      +R;
      OPN   DB [#DBpointer];
      T     DBD 4;	// = neuer Verbrauch
END_FUNCTION

FUNCTION "Transfer_Recipe" : VOID	// FC 68
TITLE = transfer recipe
//Funktion zum Übertragung der Rezeptdaten vom der Rezeptnummer entsprechenden 
//Datenbereich des Ladespeichers der CPU durch Eingabe der Rezeptnummer in der 
//OP-Maske.
//
//Function to transfer recipe datas fromm data area at load memory in PLC 
//calculated by changing recipe number in OP-mask.
AUTHOR : Fromm
VERSION : 1.1
VAR_TEMP
  T_RET_VAL : INT ;
  T_0 : DINT ;
  t_source_byte : DINT ;
  transfer : BOOL ;
  t_DB : INT ;
  t_trans1 : BOOL ;
  t_trans2 : BOOL ;
  t_trans3 : BOOL ;
  t_trans4 : BOOL ;
  t_trans5 : BOOL ;
  t_trans6 : BOOL ;
  t_trans7 : BOOL ;
  t_trans8 : BOOL ;
END_VAR
BEGIN
NETWORK
TITLE = Lokalvariabele initialisieren
      L     0;
      T     #T_0;
NETWORK
TITLE = transfer recipe start 1
// (network holds code this reader does not know; not shown)
NETWORK
TITLE = transfer recipe start 2
// (network holds code this reader does not know; not shown)
NETWORK
TITLE = transfer recipe start 3
// (network holds code this reader does not know; not shown)
NETWORK
TITLE = transfer recipe start 4
// (network holds code this reader does not know; not shown)
NETWORK
TITLE = transfer recipe start 5
// (network holds code this reader does not know; not shown)
NETWORK
TITLE = transfer recipe start 6
// (network holds code this reader does not know; not shown)
NETWORK
TITLE = transfer recipe start 7
// (network holds code this reader does not know; not shown)
NETWORK
TITLE = transfer recipe start 8
// (network holds code this reader does not know; not shown)
END_FUNCTION

FUNCTION "del_ins_line" : VOID	// FC 70
VERSION : 0.1
VAR_TEMP
  old_ptr : DINT ;
  new_ptr : DINT ;
  lp1_ctr : INT ;
  lp2_ctr : INT ;
  max_data : INT ;	//Maximale Anzahl Datensätze
  max_array : INT ;	//Größe eines Datensatzes
END_VAR
BEGIN
NETWORK
TITLE =
      L     0;
      L     "HMI_DB".rez_line;
      ==I;
      BEC;
NETWORK
TITLE = Zeile löschen
// Zu bearbeitende Zeile:db23.dbw12
//Zeile löschen db23.dbx0.6
// Zeile einfügen db23.dbx0.7
      AN    "HMI_DB".del_line;
      JC    einf;
      L     "HMI_DB".rez_line;
      L     "init_DB".max_step;
      ==I;
      JC    last;
      L     "HMI_DB".rez_line;
      DEC   1;
      L     "init_DB".step_size;
      *D;
      SLD   3;
      T     #new_ptr;
      L     "init_DB".step_size;
      SLD   3;
      L     #new_ptr;
      +D;
      T     #old_ptr;
      L     "init_DB".max_step;
      L     "HMI_DB".rez_line;
      -I;
lp2:  T     #lp2_ctr;
      L     "init_DB".step_size;
lp1:  T     #lp1_ctr;
      OPN   "RecDB";
      L     DBB [#old_ptr];
      T     DBB [#new_ptr];
      L     #new_ptr;
      L     P#1.0;
      +D;
      T     #new_ptr;
      L     #old_ptr;
      L     P#1.0;
      +D;
      T     #old_ptr;
      L     #lp1_ctr;
      LOOP  lp1;
      L     #lp2_ctr;
      LOOP  lp2;
//letzte Zeile löschen
last: L     "init_DB".max_step;
      DEC   1;
      L     "init_DB".step_size;
      *D;
      SLD   3;
      T     #new_ptr;
      L     "init_DB".step_size;
      OPN   "RecDB";
lp0:  T     #lp1_ctr;
      L     0;
      T     DBB [#new_ptr];
      L     #new_ptr;
      L     P#1.0;
      +D;
      T     #new_ptr;
      L     #lp1_ctr;
      LOOP  lp0;
      SET;
      R     "HMI_DB".del_line;
NETWORK
TITLE = Zeile einfügen
// Zu bearbeitende Zeile:db23.dbw12
// Zeile einfügen db23.dbx0.7
einf: AN    "HMI_DB".ins_line;
      JC    end;
      L     "HMI_DB".rez_line;
      L     "init_DB".max_step;
      ==I;
      JC    end1;	// nach letzter Zeile kein Einfügen möglich
      L     "init_DB".max_step;
      DEC   1;
      L     "init_DB".step_size;
      *D;
      SLD   3;
      T     #new_ptr;
      OPN   "RecDB";
      L     DBW [#new_ptr];
      L     0;
      <>I;
      JC    end1;	// Kein Einfügen möglich weil letzte Zeile belegt
      L     "init_DB".max_step;
      L     "init_DB".step_size;
      *D;
      DEC   1;
      SLD   3;
      T     #new_ptr;
      L     "init_DB".step_size;
      SLD   3;
      L     #new_ptr;
      TAK;
      -D;
      T     #old_ptr;
      L     "init_DB".max_step;
      L     "HMI_DB".rez_line;
      -I;
lp4:  T     #lp2_ctr;
      L     "init_DB".step_size;
lp3:  T     #lp1_ctr;
      OPN   "RecDB";
      L     DBB [#old_ptr];
      T     DBB [#new_ptr];
      L     #new_ptr;
      L     P#1.0;
      -D;
      T     #new_ptr;
      L     #old_ptr;
      L     P#1.0;
      -D;
      T     #old_ptr;
      L     #lp1_ctr;
      LOOP  lp3;
      L     #lp2_ctr;
      LOOP  lp4;
//eigefügte Zeile löschen
      L     "HMI_DB".rez_line;
      DEC   1;
      L     "init_DB".step_size;
      *D;
      SLD   3;
      T     #new_ptr;
      L     "init_DB".step_size;
      OPN   "RecDB";
lp5:  T     #lp1_ctr;
      L     0;
      T     DBB [#new_ptr];
      L     #new_ptr;
      L     P#1.0;
      +D;
      T     #new_ptr;
      L     #lp1_ctr;
      LOOP  lp5;
end1: SET;
      R     "HMI_DB".ins_line;
end:  NOP   0;
END_FUNCTION

FUNCTION "Hand_OP_FC" : VOID	// FC 81
VERSION : 0.1
VAR_TEMP
  loop_ctr : INT ;
  DB_ptr : INT ;
  disc_ptr : DINT ;
  err_sum : DINT ;
  err_ptr : DINT ;
  quit_ptr : DINT ;
  err_length : INT ;
  quit_length : INT ;
  t_Ret_Val : INT ;
  t_DT : DATE_AND_TIME ;
  err_ptr2 : DINT ;
  quit_ptr2 : DINT ;
  err_length2 : INT ;
  quit_length2 : INT ;
  loop_ctr2 : INT ;
END_VAR
BEGIN
NETWORK
TITLE = picture emgergency
      A     "Flag_E-Stop";
      FP    "Flag_FP81.0";
      JCN   E_on;
      L     15;
      T     "HMI_Interf".Auftrag.Par1;
      L     0;
      T     "HMI_Interf".Auftrag.Par3;
      L     51;
      T     "HMI_Interf".Auftrag.Nr;
E_on: NOP   0;
NETWORK
TITLE = check on error gravimet
      A     "fault_G";
      FP    "Flag_FP201.6";
      A     "Auto_DB".automatic;	//Störung aufgetreten
      S     "Fault_exists";
NETWORK
TITLE = read, set date and time
      CALL  "READ_CLK" (
           RET_VAL                  := #t_Ret_Val,
           CDT                      := "Clock_DB".DT_AKT);
      AN    "Clock_DB".DT_UEBERNEHMEN;
      JC    NOCL;
      CALL  "SET_CLK" (
           PDT                      := "Clock_DB".DT_NEU,
           RET_VAL                  := #t_Ret_Val);
      A     "Clock_DB".DT_UEBERNEHMEN;
      R     "Clock_DB".DT_UEBERNEHMEN;
NOCL: NOP   0;
NETWORK
TITLE = transfer datas to BR_DB gravimet
      A     "Auto_DB".automatic;
      FN    "Flag_FN202.7";
      JCN   papi;
//Date and time -> CP
      CALL  "DB_Transfer" (
           SOURCE_DB                := 2,
           SOURCE_BYTE              := L#8,
           DRAIN_DB                 := "HMI_DB".CP_DB_WRITE,
           DRAIN_BYTE               := L#8,
           LENGTH                   := 8,
           R_VAL                    := "HMI_DB".blk_ret_val);
      CALL  "DB_Transfer" (
           SOURCE_DB                := "HMI_DB".CP_DB_WRITE,
           SOURCE_BYTE              := L#0,
           DRAIN_DB                 := 124,
           DRAIN_BYTE               := L#0,
           LENGTH                   := 280,
           R_VAL                    := "HMI_DB".blk_ret_val);
      L     "HMI_DB".print;
      L     0;	//kein Ausdruck
      ==I;
      JC    ndr;
      A(;
      L     "HMI_DB".print;
      L     2;	//Druck nur bei Störung
      ==I;
      );
      JC    derr;
      A     "Fault_exists";
      JCN   ndr;
derr: AN    "HMI_DB".print_BR;	//Wertänderung Druckanstoß
      =     "HMI_DB".print_BR;
ndr:  A     "Fault_exists";
      R     "Fault_exists";
papi: NOP   0;
NETWORK
TITLE = add filling to tank
      L     "init_DB".highest_comp;
M002: T     #loop_ctr;
      L     30;
      +I;
      T     #DB_ptr;
      OPN   DB [#DB_ptr];
      L     DBD 0;	// Tankinhalt
      L     DBD 40;	// Füllung
      +R;
      T     DBD 0;
      L     0;
      T     DBD 40;
      L     #loop_ctr;
      LOOP  M002;
      NOP   0;
NETWORK
TITLE = clear consumption
      AN    "HMI_DB".clear_cons;
      JC    M003;
      L     "init_DB".highest_comp;
M004: T     #loop_ctr;	// Verbrauch je Komponente
      L     #loop_ctr;
      L     30;
      +I;
      T     #DB_ptr;
      OPN   DB [#DB_ptr];
      L     0;
      T     DBD 4;
      L     #loop_ctr;
      LOOP  M004;
      R     "HMI_DB".clear_cons;
M003: NOP   0;
      AN    "HMI_DB".clear_OP;
      JC    M005;
      LAR1  P#4.0;
      L     "init_DB".starts;
      OPN   "Start_DB";
M006: T     #loop_ctr;	// Vorratsverbrauch und Anzahl
      L     0;
      T     DBD [AR1,P#0.0];
      T     DBD [AR1,P#4.0];
      +AR1  P#30.0;
      L     #loop_ctr;
      LOOP  M006;
      R     "HMI_DB".clear_OP;
M005: NOP   0;
NETWORK
TITLE = Asynchronfehler
      A     DB10.DBX 48.0;	//Fehler aufgetreten
      AN    "Restart_Timer";
      A     "CV_DELAYED";
      S     DB20.DBX 75.5;
      S     "stop_G";
      A     DB11.DBX 48.0;
      AN    "Restart_Timer";
      A     "CV_DELAYED";
      S     DB20.DBX 75.6;
      S     "stop_G";
NETWORK
TITLE = Abstand der Justierpunkte
      O     DB10.DBX 55.0;
      O     DB11.DBX 55.0;
      S     DB20.DBX 72.5;
NETWORK
TITLE = Handbedienung nullen
      A     "Auto_DB".automatic;
      JC    m009;
      L     3;
      AN    "VISU".Button.zero_main_scale;
      JC    M007;
      A     "WScale1".no_zero;
      S     DB20.DBX 73.0;
      S     "WScale1".show_zero;
      JC    M007;
      T     "WScale1".Command;
      S     "WScale1".WriteCommand;
M007: AN    "VISU".Button.zero_sub_scale;
      JC    M008;
      A     "WScale2".no_zero;
      S     DB20.DBX 72.0;
      S     "WScale2".show_zero;
      JC    M008;
      T     "WScale2".Command;
      S     "WScale2".WriteCommand;
M008: NOP   0;
NETWORK
TITLE = Handbedienung tarieren/Inhalt
      A     "Auto_DB".automatic;
      JC    m009;
      A     "VISU".Button.tare_main_scale;
      S     "WScale1".TareScale;
      A     "VISU".Button.cont_main_scale;
      S     "WScale1".ClearTara;
m009: NOP   0;
END_FUNCTION

FUNCTION "comp_scale" : VOID	// FC 85
VERSION : 0.1
VAR_INPUT
  component : INT ;
END_VAR
VAR_OUTPUT
  scale_nr : INT ;
END_VAR
VAR_TEMP
  KompPointer : DINT ;
  T_AR1 : DINT ;
  T_AR2 : DINT ;
END_VAR
BEGIN
NETWORK
TITLE =
      TAR1  #T_AR1;
      TAR2  #T_AR2;
NETWORK
TITLE =
      L     0;
      L     #component;
      ==I;
      JC    nok;
      INC   9;	// Startadresse DB1-1
      SLD   3;
      T     #KompPointer;
      OPN   "init_DB";
      L     DBB [#KompPointer];
nok:  T     #scale_nr;
NETWORK
TITLE =
      LAR1  #T_AR1;
      LAR2  #T_AR2;
END_FUNCTION

FUNCTION "MPI_level_2s" : VOID	// FC 87
VERSION : 0.1
VAR_INPUT
  full : BOOL ;
  empty : BOOL ;
END_VAR
VAR_OUTPUT
  level : BYTE ;
END_VAR
BEGIN
NETWORK
TITLE =
      L     0;
      AN    "CV_DELAYED";
      JC    tran;
      L     80;
      A     "CV_DELAYED";
      AN    #full;
      JC    tran;
      L     50;
      A     #empty;
      JC    tran;
      L     10;
tran: T     #level;
END_FUNCTION

FUNCTION "Start series gravimet" : VOID	// FC 91
VERSION : 0.1
VAR_INPUT
  Sel1 : BOOL ;
  Rec1 : BOOL ;
  Sel2 : BOOL ;
  Rec2 : BOOL ;
  Sel3 : BOOL ;
  Rec3 : BOOL ;
  Sel4 : BOOL ;
  Rec4 : BOOL ;
  Sel5 : BOOL ;
  Rec5 : BOOL ;
  Sel6 : BOOL ;
  Rec6 : BOOL ;
  Sel7 : BOOL ;
  Rec7 : BOOL ;
  Sel8 : BOOL ;
  Rec8 : BOOL ;
END_VAR
VAR_OUTPUT
  Free1 : BOOL ;
  Free2 : BOOL ;
  Free3 : BOOL ;
  Free4 : BOOL ;
  Free5 : BOOL ;
  Free6 : BOOL ;
  Free7 : BOOL ;
  Free8 : BOOL ;
END_VAR
VAR_TEMP
  Startnr : INT ;
  noStart : BOOL ;
END_VAR
BEGIN
NETWORK
TITLE = Freigaben löschen
      L     DB21.DBB 8;	// remanente Starts
      L     MB 135;
      AW;
      T     MB 135;
      L     DB21.DBB 8;
      L     0;
      <>I;
      JC    go;
      L     0;
      T     "StartSeriesDB".buffer[1];
go:   NOP   0;
NETWORK
TITLE = Start 1
      A     #Sel1;
      AN    #Rec1;
      JCN   st2;
      CALL  "FFL-G" (
           Value                    := 1);
NETWORK
TITLE = Start 2
st2:  A     #Sel2;
      AN    #Rec2;
      JCN   st3;
      CALL  "FFL-G" (
           Value                    := 2);
NETWORK
TITLE = Start 3
st3:  A     #Sel3;
      AN    #Rec3;
      JCN   st4;
      CALL  "FFL-G" (
           Value                    := 3);
NETWORK
TITLE = Start 4
st4:  A     #Sel4;
      AN    #Rec4;
      JCN   st5;
      CALL  "FFL-G" (
           Value                    := 4);
NETWORK
TITLE = Start 5
st5:  A     #Sel5;
      AN    #Rec5;
      JCN   st6;
      CALL  "FFL-G" (
           Value                    := 5);
NETWORK
TITLE = Start 6
st6:  A     #Sel6;
      AN    #Rec6;
      JCN   st7;
      CALL  "FFL-G" (
           Value                    := 6);
NETWORK
TITLE = Start 7
st7:  A     #Sel7;
      AN    #Rec7;
      JCN   st8;
      CALL  "FFL-G" (
           Value                    := 7);
NETWORK
TITLE = Start 8
st8:  A     #Sel8;
      AN    #Rec8;
      JCN   st9;
      CALL  "FFL-G" (
           Value                    := 8);
NETWORK
TITLE = Ende wenn Hauptstart weg oder Start läuft
st9:  L     DB21.DBB 8;
      L     0;
      <>I;
      BEC;
      A     "main_start";
      JC    main;
      OPN   "StartSeriesDB";
      L     0;
      T     DBD 0;
      T     DBD 4;
      T     DBW 8;
      T     DBD 10;
      BEU;
main: NOP   0;
NETWORK
TITLE = Startpuffer auslesen
      CALL  "FFU-G" (
           empty                    := #noStart,
           value                    := #Startnr);
      A     #noStart;
      BEC;
NETWORK
TITLE = Freigabe für Start erteilen
      L     1;
      L     #Startnr;
      ==I;
      A     #Sel1;
      AN    #Rec1;
      S     #Free1;
      L     2;
      L     #Startnr;
      ==I;
      A     #Sel2;
      AN    #Rec2;
      S     #Free2;
      L     3;
      L     #Startnr;
      ==I;
      A     #Sel3;
      AN    #Rec3;
      S     #Free3;
      L     4;
      L     #Startnr;
      ==I;
      A     #Sel4;
      AN    #Rec4;
      S     #Free4;
      L     5;
      L     #Startnr;
      ==I;
      A     #Sel5;
      AN    #Rec5;
      S     #Free5;
      L     6;
      L     #Startnr;
      ==I;
      A     #Sel6;
      AN    #Rec6;
      S     #Free6;
      L     7;
      L     #Startnr;
      ==I;
      A     #Sel7;
      AN    #Rec7;
      S     #Free7;
      L     8;
      L     #Startnr;
      ==I;
      A     #Sel8;
      AN    #Rec8;
      S     #Free8;
END_FUNCTION

FUNCTION "FFL-G" : VOID	// FC 92
TITLE = FiFo-Speicher laden
VERSION : 0.1
VAR_INPUT
  Value : INT ;
END_VAR
BEGIN
NETWORK
TITLE = Startpuffer öffnen
      OPN   "StartSeriesDB";
NETWORK
TITLE = Start schon im Puffer?
      L     DBB 0;
      L     #Value;
      ==I;
      BEC;
      L     DBB 1;
      L     #Value;
      ==I;
      BEC;
      L     DBB 2;
      L     #Value;
      ==I;
      BEC;
      L     DBB 3;
      L     #Value;
      ==I;
      BEC;
      L     DBB 4;
      L     #Value;
      ==I;
      BEC;
      L     DBB 5;
      L     #Value;
      ==I;
      BEC;
      L     DBB 6;
      L     #Value;
      ==I;
      BEC;
      L     DBB 7;
      L     #Value;
      ==I;
      BEC;
      L     DBB 8;
      L     #Value;
      ==I;
      BEC;
NETWORK
TITLE = Pointer erhöhen, Wert in Puffer
      L     DBD 10;
      L     P#7.0;
      >D;
      BEC;	// Puffer bereits voll
      L     DBD 10;
      INC   8;
      T     DBD 10;
      L     #Value;
      T     DBB [DBD 10];
END_FUNCTION

FUNCTION "FFU-G" : VOID	// FC 93
TITLE = FiFo-Speicher auslesen
VERSION : 0.1
VAR_OUTPUT
  empty : BOOL ;
  value : INT ;
END_VAR
BEGIN
NETWORK
TITLE = Test ob was im Puffer steht
      L     0;
      T     #value;
      L     "StartSeriesDB".ptr;
      L     0;
      ==D;
      =     #empty;
      BEC;
NETWORK
TITLE = Werte nachrücken
      L     DBD 0;
      SLD   8;
      T     DBD 0;
      L     DBD 3;
      SLD   8;
      T     DBD 3;
      L     DBD 6;
      SLD   8;
      T     DBD 6;
NETWORK
TITLE = Wert auslesen
      L     DBB 0;
      T     #value;
NETWORK
TITLE = Pointer erniedrigen
      L     DBD 10;
      DEC   8;
      T     DBD 10;
END_FUNCTION

FUNCTION "FC_SET_BIT" : VOID	// FC 110
VERSION : 0.1
VAR_INPUT
  RUN_BIT : BOOL ;	//Bit für Visualisierung das gesetzt werden soll
  ERR_BIT : BOOL ;
END_VAR
VAR_OUTPUT
  VISU_BYTE : BYTE ;	//Byte für Visualisierung in dem Bits gesetzt werden sollen
END_VAR
VAR_TEMP
  t_RUN_BIT : BOOL ;
  t_ERR_BIT : BOOL ;
END_VAR
BEGIN
NETWORK
TITLE =
      L     0;
      T     LB 0;
      A     #ERR_BIT;
      =     #t_ERR_BIT;
      A     #RUN_BIT;
      =     #t_RUN_BIT;
      L     LB 0;
      T     #VISU_BYTE;
END_FUNCTION

FUNCTION "DT_Transfer" : VOID	// FC 166
VERSION : 0.1
VAR_INPUT
  br_db_quelle : WORD ;
  br_db_ziel : WORD ;
END_VAR
VAR_TEMP
  t_br_db_quelle : WORD ;
  t_br_db_ziel : WORD ;
  t_loop : INT ;
END_VAR
BEGIN
NETWORK
TITLE =
      L     #br_db_quelle;
      T     #t_br_db_quelle;
      L     #br_db_ziel;
      T     #t_br_db_ziel;
      OPN   DB [#t_br_db_quelle];
      L     DBD 8;
      OPN   DB [#t_br_db_ziel];
      T     DBD 8;
      OPN   DB [#t_br_db_quelle];
      L     DBD 12;
      OPN   DB [#t_br_db_ziel];
      T     DBD 12;
END_FUNCTION

FUNCTION "DB_Transfer" : VOID	// FC 167
VERSION : 0.1
VAR_INPUT
  SOURCE_DB : INT ;	//Data Block Source - Datenbausteinnr. Quelle
  SOURCE_BYTE : DINT ;	//First Byte Source - Erstes Byte Quelle
  DRAIN_DB : INT ;	//Data Block Drain - Datenbausteinnr. Ziel
  DRAIN_BYTE : DINT ;	//First Byte Ziel - Erstes Byte Ziel
  LENGTH : INT ;	//Length of Datas in BYTE - Datenlänge in BYTE
END_VAR
VAR_OUTPUT
  R_VAL : INT ;	//RET_VAL of SFC20
END_VAR
VAR_TEMP
  ANY_SOURCE : ANY ;
  ANY_DRAIN : ANY ;
  stack1 : DINT ;
END_VAR
BEGIN
NETWORK
TITLE = Save Registers - Adressregister retten
      TAR1  #stack1;
NETWORK
TITLE =
      LAR1  P##ANY_SOURCE;	// Start address source
      L     W#16#1002;	// Syntax-ID STEP 7)    Source type BYTE
      T     LW [AR1,P#0.0];
      L     #LENGTH;	// Length of Datas
      T     LW [AR1,P#2.0];
      L     #SOURCE_DB;	// Nr of Source DB
      T     LW [AR1,P#4.0];
      L     P#DBX 0.0;	// Data Type DB
      L     #SOURCE_BYTE;	// Start Byte
      SLD   3;
      +D;
      T     LD [AR1,P#6.0];
NETWORK
TITLE =
      LAR1  P##ANY_DRAIN;	// Start address source
      L     W#16#1002;	// Syntax-ID STEP 7)    Source type BYTE
      T     LW [AR1,P#0.0];
      L     #LENGTH;	// Length of Datas
      T     LW [AR1,P#2.0];
      L     #DRAIN_DB;	// Nr of Source DB
      T     LW [AR1,P#4.0];
      L     P#DBX 0.0;	// Data Type DB
      L     #DRAIN_BYTE;	// Start Byte
      SLD   3;
      +D;
      T     LD [AR1,P#6.0];
NETWORK
TITLE =
      CALL  "BLKMOV" (
           SRCBLK                   := #ANY_SOURCE,
           RET_VAL                  := #R_VAL,
           DSTBLK                   := #ANY_DRAIN);
NETWORK
TITLE = Restore Registers -Adressregister wieder herstellen
      LAR1  #stack1;
END_FUNCTION

FUNCTION "Rec_handling" : VOID	// FC 190
TITLE = handling recipe
//Dieser Baustein dient zur Verwaltung von Rezepten im Ladespeicher der CPU. 
//Hierzu müssen Datenbausteine mit der Option "unlinked" ab DB333 angelegt sein. 
//In diesen Datenbausteinen können, aufgrund der maximalen Datenbausteingröße der 
//CPU 315, jeweils 50 Rezepte gespeichert werden. Das 
//heißt im DB 333 die Rezepte 1-50, im DB 334 die Rezepte 51-100 und so weiter.
//
//This function handles recipes saved in load memory of the PLC. Therefore the 
//data blocks from DB 333 must be created with the option "unlinked". Each DB 
//contains, because the DB-dimension of PLC315, 50 recipes seams like DB 333 
//contains recipes 1-50, DB 334 contains recipes 51-100 and so on.
AUTHOR : Fromm
VERSION : 1.0
VAR_TEMP
  t_source_byte : DINT ;
  t_ret_val : INT ;
  t_drain_byte : DINT ;
  t_t0 : INT ;
  t_rec_DB : INT ;
  t_DB : INT ;
  t_read : BOOL ;
  t_busy : BOOL ;
  t_no_comp : BOOL ;
END_VAR
BEGIN
NETWORK
TITLE = transfer recipe to DB22
//Der Datenbaustein 22 dient zur Bearbeitung der Rezepte am Bediengerät. Hierzu 
//wird in diesem Netzwerk der dem Rezept entsprechende Datenbereich aus dem 
//entsprechenden Datenbaustein im Ladespeicher geholt und in den DB 22 
//geschrieben.
//
//Manipulation of recipes at the human-machine-interface was supported by 
//datablock 22. Therefore the datas must be read from the data block, at loading 
//memory in the PLC, calculated throuh recipe number and writen to data block 22.
// (network holds code this reader does not know; not shown)
//Zeit muss verlängert werden damit das MP370 die Varialbe sicher lesen kann
//Zeit muss verlängert werden damit das MP370 die Varialbe sicher lesen kann
//Da der gleiche FC zwei mal aufgerufen wird muss sicher gestellt werden,
//das der erste FC vollständig abgearbeitet ist bevors zum nachsten Aufruf geht.
NETWORK
TITLE = save recipe to DB
//In diesem Netzwerk wird der bearbeitete DB 22 in den der Rezeptnummer 
//entsprechenden Datenbereich des entsprechenden Datenbausteins im 
//Ladespeicher der CPU geschrieben.
//
//The manipulated data block 22 will be writen into data block, calculated by 
//recipe number, at load memory in the PLC.
// (network holds code this reader does not know; not shown)
//Rezept löschen sperren
//Rezept überschreiben
//    R     "RecDB".busy_save
//Wenn Nein gedrückt wird oder anderes Rezept ausgewählt wird (am MP370)
//Änderungen sind abgespeichert
NETWORK
TITLE = update recipe start 1
//Beim Speichern eines Rezeptes wird hier überprüft ob dieses im Start 1 
//verwendet 
//wird. Wenn ja dann wird dieses auch in den für den Start 1 verantwortlichen 
//DB150 geschrieben.
//
//If the saved recipe runs at start 1 it was saved in the DB150 too.
      A     M 190.1;
      JC    nosp;
      L     "Start_DB".Start[1].Rezept;
      L     "RecDB".rec_new;
      ==I;
      JCN   no1;
      L     0;
      T     "Start_DB".Start[1].Rezept_alt;
NETWORK
TITLE = update recipe start 2
//Beim Speichern eines Rezeptes wird hier überprüft ob dieses im Start 2 
//verwendet 
//wird. Wenn ja dann wird dieses auch in den für den Start 2 verantwortlichen 
//DB151 geschrieben.
//
//If the saved recipe runs at start 2 it was saved in the DB151 too.
no1:  L     "Start_DB".Start[2].Rezept;
      L     "RecDB".rec_new;
      ==I;
      JCN   no2;
      L     0;
      T     "Start_DB".Start[2].Rezept_alt;
NETWORK
TITLE = update recipe start 3
//Beim Speichern eines Rezeptes wird hier überprüft ob dieses im Start 3 
//verwendet 
//wird. Wenn ja dann wird dieses auch in den für den Start 3 verantwortlichen 
//DB152 geschrieben.
//
//If the saved recipe runs at start 3 it was saved in the DB152 too.
no2:  L     "Start_DB".Start[3].Rezept;
      L     "RecDB".rec_new;
      ==I;
      JCN   no3;
      L     0;
      T     "Start_DB".Start[3].Rezept_alt;
NETWORK
TITLE = update recipe start 4
//Beim Speichern eines Rezeptes wird hier überprüft ob dieses im Start 4 
//verwendet 
//wird. Wenn ja dann wird dieses auch in den für den Start 4 verantwortlichen 
//DB153 geschrieben.
//
//If the saved recipe runs at start 4 it was saved equal in the DB153 too.
no3:  L     "Start_DB".Start[4].Rezept;
      L     "RecDB".rec_new;
      ==I;
      JCN   no4;
      L     0;
      T     "Start_DB".Start[4].Rezept_alt;
NETWORK
TITLE = update recipe start 5
//Beim Speichern eines Rezeptes wird hier überprüft ob dieses im Start 5 
//verwendet 
//wird. Wenn ja dann wird dieses auch in den für den Start 5 verantwortlichen 
//DB154 geschrieben.
//
//If the saved recipe runs at start 5 it was saved equal in the DB154 too.
no4:  L     "Start_DB".Start[5].Rezept;
      L     "RecDB".rec_new;
      ==I;
      JCN   no5;
      L     0;
      T     "Start_DB".Start[5].Rezept_alt;
NETWORK
TITLE = update recipe start 6
//Beim Speichern eines Rezeptes wird hier überprüft ob dieses im Start 6 
//verwendet 
//wird. Wenn ja dann wird dieses auch in den für den Start 6 verantwortlichen 
//DB155 geschrieben.
//
//If the saved recipe runs at start 6 it was saved equal in the DB155 too.
no5:  L     "Start_DB".Start[6].Rezept;
      L     "RecDB".rec_new;
      ==I;
      JCN   no6;
      L     0;
      T     "Start_DB".Start[6].Rezept_alt;
NETWORK
TITLE = update recipe start 7
//Beim Speichern eines Rezeptes wird hier überprüft ob dieses im Start 7 
//verwendet 
//wird. Wenn ja dann wird dieses auch in den für den Start 7 verantwortlichen 
//DB156 geschrieben.
//
//If the saved recipe runs at start 7 it was saved equal in the DB156 too.
no6:  L     "Start_DB".Start[7].Rezept;
      L     "RecDB".rec_new;
      ==I;
      JCN   no7;
      L     0;
      T     "Start_DB".Start[7].Rezept_alt;
NETWORK
TITLE = update recipe start 8
//Beim Speichern eines Rezeptes wird hier überprüft ob dieses im Start 8 
//verwendet 
//wird. Wenn ja dann wird dieses auch in den für den Start 8 verantwortlichen 
//DB157 geschrieben.
//
//If the saved recipe runs at start 8 it was saved equal in the DB157 too.
no7:  L     "Start_DB".Start[8].Rezept;
      L     "RecDB".rec_new;
      ==I;
      JCN   nosp;
      L     0;
      T     "Start_DB".Start[8].Rezept_alt;
nosp: NOP   0;
NETWORK
TITLE = delete recipe
//Mit diesem Netzwerk werden Rezepte gelöscht. Das heißt der DB 22 wird mit 0 
//beschrieben und in den der Rezeptnummer entsprechenden Datenbereich des 
//entsprechenden Datenbausteins im Ladespeicher der CPU geschrieben.
//
//To delete a recipe the data block 22 must be overwrite with 0 and saved at the 
//data block, calculated by recipe number, at load memory in the PLC.
// (network holds code this reader does not know; not shown)
NETWORK
TITLE = copy recipe
//Dieses Netzwerk dient zum kopieren von Rezepten. Hierzu wird das im DB22 
//befindliche Rezept in den DB 122 geschrieben.
//
//To copy a recipe read data block 22 an write the datas into data block 
//122(buffer).
      AN    "RecDB".rec_copy;
      JC    ncop;
      CALL  "DB_Transfer" (
           SOURCE_DB                := 22,
           SOURCE_BYTE              := L#0,
           DRAIN_DB                 := 122,
           DRAIN_BYTE               := L#0,
           LENGTH                   := 250,
           R_VAL                    := #t_ret_val);
      R     "RecDB".rec_copy;
ncop: NOP   0;
NETWORK
TITLE = paste recipe
//In diesem Netzwerk wird das, durch kopieren im DB122 befindliche, Rezept in den 
//DB 22 geschrieben.
//
//To paste a recipe read data block 122(buffer) and write the datas into data 
//block 22.
      AN    "RecDB".rec_paste;
      JC    npa;
      CALL  "DB_Transfer" (
           SOURCE_DB                := 122,
           SOURCE_BYTE              := L#0,
           DRAIN_DB                 := 22,
           DRAIN_BYTE               := L#0,
           LENGTH                   := 250,
           R_VAL                    := #t_ret_val);
      R     "RecDB".rec_paste;
npa:  NOP   0;
END_FUNCTION

FUNCTION "DB_compare" : VOID	// FC 191
VERSION : 0.1
VAR_INPUT
  DB_Nr1 : INT ;
  Start_DB1 : INT ;
  DB_Nr2 : INT ;
  Start_DB2 : INT ;
  Laenge_DBW : INT ;
END_VAR
VAR_OUTPUT
  result : BOOL ;
END_VAR
VAR_TEMP
  adr1 : DWORD ;
  DB_1 : WORD ;
  DB_2 : WORD ;
  Loop : WORD ;
  adr2 : DWORD ;
END_VAR
BEGIN
NETWORK
TITLE =
      L     #Start_DB1;
      SLW   3;	// Pointer adaptation
      T     #adr1;
      L     #Start_DB2;
      SLW   3;
      T     #adr2;
      L     #DB_Nr1;	// DB1 load
      T     #DB_1;
      L     #DB_Nr2;	// DB2 load
      T     #DB_2;
      L     #Laenge_DBW;	// Number of DB words to be compared
JMP1: T     #Loop;
      OPN   DB [#DB_1];
      L     DBW [#adr1];
      OPN   DB [#DB_2];
      L     DBW [#adr2];
      <>I;
      JC    JMP2;
      L     #adr1;
      L     16;	// add 2
      +D;
      T     #adr1;
      L     #adr2;
      L     16;
      +D;
      T     #adr2;
      CLR;	// set result = 0
      =     #result;
      L     #Loop;
      LOOP  JMP1;
      BEU;
JMP2: NOP   0;
      SET;
      =     #result;
END_FUNCTION

// FC 200: know-how protected block, not included

FUNCTION "read_load_memory" : VOID	// FC 267
TITLE = read data block area from load memory
//Funktion zum Lesen eines Datenbausteinbereiches aus dem Ladespeicher der CPU.
//
//Function to read a data blok area from load memory of PLC.
VERSION : 0.1
VAR_INPUT
  SOURCE_DB : INT ;	//Data Block Source - Datenbausteinnr. Quelle
  SOURCE_BYTE : DINT ;	//First Byte Source - Erstes Byte Quelle
  DRAIN_DB : INT ;	//Data Block Drain - Datenbausteinnr. Ziel
  DRAIN_BYTE : DINT ;	//First Byte Ziel - Erstes Byte Ziel
  LENGTH : INT ;	//Length of Datas in BYTE - Datenlänge in BYTE
  i_read : BOOL ;
END_VAR
VAR_OUTPUT
  R_VAL : INT ;	//RET_VAL of SFC20
  o_busy : BOOL ;
END_VAR
VAR_TEMP
  ANY_SOURCE : ANY ;
  ANY_DRAIN : ANY ;
  stack1 : DINT ;
END_VAR
BEGIN
NETWORK
TITLE = Save Registers - Adressregister retten
      TAR1  #stack1;
NETWORK
TITLE =
      LAR1  P##ANY_SOURCE;	// Start address source
      L     W#16#1002;	// Syntax-ID STEP 7)    Source type BYTE
      T     LW [AR1,P#0.0];
      L     #LENGTH;	// Length of Datas
      T     LW [AR1,P#2.0];
      L     #SOURCE_DB;	// Nr of Source DB
      T     LW [AR1,P#4.0];
      L     P#DBX 0.0;	// Data Type DB
      L     #SOURCE_BYTE;	// Start Byte
      SLD   3;
      +D;
      T     LD [AR1,P#6.0];
NETWORK
TITLE =
      LAR1  P##ANY_DRAIN;	// Start address source
      L     W#16#1002;	// Syntax-ID STEP 7)    Source type BYTE
      T     LW [AR1,P#0.0];
      L     #LENGTH;	// Length of Datas
      T     LW [AR1,P#2.0];
      L     #DRAIN_DB;	// Nr of Source DB
      T     LW [AR1,P#4.0];
      L     P#DBX 0.0;	// Data Type DB
      L     #DRAIN_BYTE;	// Start Byte
      SLD   3;
      +D;
      T     LD [AR1,P#6.0];
NETWORK
TITLE =
      CALL  "READ_DBL" (
           REQ                      := #i_read,
           SRCBLK                   := #ANY_SOURCE,
           RET_VAL                  := #R_VAL,
           BUSY                     := #o_busy,
           DSTBLK                   := #ANY_DRAIN);
NETWORK
TITLE = Restore Registers -Adressregister wieder herstellen
      LAR1  #stack1;
END_FUNCTION

FUNCTION "write_load_memory" : VOID	// FC 268
TITLE = write data block area to load memory
//Funktion zum Schreiben eines Datenbausteinbereiches in den Ladespeicher der CPU.
//
//Function to write a data block area into load memory of PLC.
VERSION : 0.1
VAR_INPUT
  SOURCE_DB : INT ;	//Data Block Source - Datenbausteinnr. Quelle
  SOURCE_BYTE : DINT ;	//First Byte Source - Erstes Byte Quelle
  DRAIN_DB : INT ;	//Data Block Drain - Datenbausteinnr. Ziel
  DRAIN_BYTE : DINT ;	//First Byte Ziel - Erstes Byte Ziel
  LENGTH : INT ;	//Length of Datas in BYTE - Datenlänge in BYTE
  i_write : BOOL ;
END_VAR
VAR_OUTPUT
  R_VAL : INT ;	//RET_VAL of SFC20
  o_busy : BOOL ;
END_VAR
VAR_TEMP
  ANY_SOURCE : ANY ;
  ANY_DRAIN : ANY ;
  stack1 : DINT ;
END_VAR
BEGIN
NETWORK
TITLE = Save Registers - Adressregister retten
      TAR1  #stack1;
NETWORK
TITLE =
      LAR1  P##ANY_SOURCE;	// Start address source
      L     W#16#1002;	// Syntax-ID STEP 7)    Source type BYTE
      T     LW [AR1,P#0.0];
      L     #LENGTH;	// Length of Datas
      T     LW [AR1,P#2.0];
      L     #SOURCE_DB;	// Nr of Source DB
      T     LW [AR1,P#4.0];
      L     P#DBX 0.0;	// Data Type DB
      L     #SOURCE_BYTE;	// Start Byte
      SLD   3;
      +D;
      T     LD [AR1,P#6.0];
NETWORK
TITLE =
      LAR1  P##ANY_DRAIN;	// Start address source
      L     W#16#1002;	// Syntax-ID STEP 7)    Source type BYTE
      T     LW [AR1,P#0.0];
      L     #LENGTH;	// Length of Datas
      T     LW [AR1,P#2.0];
      L     #DRAIN_DB;	// Nr of Source DB
      T     LW [AR1,P#4.0];
      L     P#DBX 0.0;	// Data Type DB
      L     #DRAIN_BYTE;	// Start Byte
      SLD   3;
      +D;
      T     LD [AR1,P#6.0];
NETWORK
TITLE =
      CALL  "WRIT_DBL" (
           REQ                      := #i_write,
           SRCBLK                   := #ANY_SOURCE,
           RET_VAL                  := #R_VAL,
           BUSY                     := #o_busy,
           DSTBLK                   := #ANY_DRAIN);
NETWORK
TITLE = Restore Registers -Adressregister wieder herstellen
      LAR1  #stack1;
END_FUNCTION

DATA_BLOCK "init_DB"	// DB 1
VERSION : 0.1
  STRUCT
   max_step : INT  := 10;
   step_size : INT  := 10;
   max_scale : INT  := 2;
   colour_starts : BYTE ;
   highest_comp : INT  := 32;
   comp_scale : ARRAY  [1 .. 50 ] OF BYTE ;
   max_recipe : INT  := 200;
   starts : INT  := 8;
   CP_DB_MIN : WORD ;	//Zeiger auf den ersten CP-DB
   CP_DB_ANZ : WORD ;	//Zeiger auf den letzten CP-DB
   CP_DB_MIN_P : WORD ;	//Zeiger auf den ersten CP-DB
   CP_DB_ANZ_P : WORD ;	//Zeiger auf den letzten CP-DB
  END_STRUCT ;	
BEGIN
   max_step := 24;
   step_size := 10;
   max_scale := 3;
   highest_comp := 17;
   comp_scale[1] := B#16#1;
   comp_scale[2] := B#16#1;
   comp_scale[3] := B#16#1;
   comp_scale[4] := B#16#1;
   comp_scale[5] := B#16#FF;
   comp_scale[6] := B#16#2;
   comp_scale[7] := B#16#2;
   comp_scale[8] := B#16#2;
   comp_scale[9] := B#16#2;
   comp_scale[10] := B#16#2;
   comp_scale[11] := B#16#2;
   comp_scale[12] := B#16#3;
   comp_scale[13] := B#16#3;
   comp_scale[14] := B#16#3;
   comp_scale[15] := B#16#3;
   comp_scale[16] := B#16#3;
   comp_scale[17] := B#16#3;
   max_recipe := 200;
   starts := 3;
   CP_DB_MIN := W#16#A0;
   CP_DB_ANZ := W#16#A;
   CP_DB_MIN_P := W#16#AA;
   CP_DB_ANZ_P := W#16#A;
END_DATA_BLOCK

DATA_BLOCK "Clock_DB"	// DB 2
VERSION : 0.1
  STRUCT
   DT_NEU : DATE_AND_TIME ;
   DT_AKT : DATE_AND_TIME ;
   DT_RES01 : BYTE ;
   DT_RES02 : BYTE ;
   DT_RES03 : BYTE ;
   DT_RES04 : BYTE ;
   DT_UEBERNEHMEN : BOOL ;
   RES16_1 : BOOL ;
   RES16_2 : BOOL ;
   RES16_3 : BOOL ;
   RES16_4 : BOOL ;
   RES16_5 : BOOL ;
   RES16_6 : BOOL ;
   RES16_7 : BOOL ;
   RES17_0 : BOOL ;
   RES17_1 : BOOL ;
   RES17_2 : BOOL ;
   RES17_3 : BOOL ;
   RES17_4 : BOOL ;
   RES17_5 : BOOL ;
   RES17_6 : BOOL ;
   RES17_7 : BOOL ;
  END_STRUCT ;	
BEGIN
END_DATA_BLOCK

DATA_BLOCK "VISU"	// DB 3
VERSION : 0.1
  STRUCT
   Button : STRUCT 	//Taster in Visualisierung
    Auto : BOOL ;
    Start : BOOL ;
    Stop : BOOL ;
    Quit : BOOL ;
    horn_off : BOOL ;
    continuous_run : BOOL ;
    lamp_test : BOOL ;
    res3 : BOOL ;
    SelStart1 : BOOL ;
    SelStart2 : BOOL ;
    SelStart3 : BOOL ;
    SelStart4 : BOOL ;
    SelStart5 : BOOL ;
    SelStart6 : BOOL ;
    SelStart7 : BOOL ;
    SelStart8 : BOOL ;
    RW_V1 : BOOL ;
    RW_V2 : BOOL ;
    RW_V3 : BOOL ;
    RW_V3_FASTSLOW : BOOL ;
    RW_V5 : BOOL ;
    RW_V6 : BOOL ;
    RW_V7 : BOOL ;
    RW_LW : BOOL ;
    RW_HW : BOOL ;
    start_lacquer : BOOL ;
    stop_lacquer : BOOL ;
    cont_run_lacquer : BOOL ;
    auto_lacquer : BOOL ;
    res45 : BOOL ;
    res46 : BOOL ;
    Entl_SW : BOOL ;	//Entleeren Subwaage
    Entl_HW_V1 : BOOL ;	//Entleeren Hauptwaage in Vorrat 1
    Entl_HW_V2 : BOOL ;	//Entleeren Hauptwaage in Vorrat 1
    Entl_HW_V3 : BOOL ;	//Entleeren Hauptwaage in Vorrat 1
    Entl_HW_V4 : BOOL ;	//Entleeren Hauptwaage in Vorrat 1
    Entl_HW_V5 : BOOL ;	//Entleeren Hauptwaage in Vorrat 1
    Entl_HW_V6 : BOOL ;	//Entleeren Hauptwaage in Vorrat 1
    Entl_HW_V7 : BOOL ;	//Entleeren Hauptwaage in Vorrat 1
    Entl_FW : BOOL ;	//Entleeren Hauptwaage in Vorrat 1
    dosi_C1 : BOOL ;
    dosi_C2 : BOOL ;
    dosi_C3 : BOOL ;
    dosi_C4 : BOOL ;
    dosi_C5 : BOOL ;
    dosi_C6_ms : BOOL ;
    dosi_C6_ss : BOOL ;
    dosi_C7 : BOOL ;
    dosi_C8 : BOOL ;
    dosi_C9 : BOOL ;
    dosi_C10 : BOOL ;
    dosi_C11 : BOOL ;
    dosi_C12 : BOOL ;
    dosi_C13 : BOOL ;
    dosi_C14 : BOOL ;
    dosi_C15 : BOOL ;
    dosi_C16 : BOOL ;
    dosi_C17 : BOOL ;
    dosi_C18 : BOOL ;
    dosi_C19 : BOOL ;
    dosi_C20 : BOOL ;
    dosi_C21 : BOOL ;
    dosi_C22 : BOOL ;
    dosi_C23 : BOOL ;
    dosi_C24 : BOOL ;
    dosi_C25 : BOOL ;
    dosi_C26 : BOOL ;
    dosi_C27 : BOOL ;
    dosi_C28 : BOOL ;
    dosi_C29 : BOOL ;
    dosi_C30 : BOOL ;
    dosi_C31 : BOOL ;
    dosi_C32 : BOOL ;
    c27_circ : BOOL ;
    res52 : BOOL ;
    res53 : BOOL ;
    res54 : BOOL ;
    res55 : BOOL ;
    res56 : BOOL ;
    res57 : BOOL ;
    zero_main_scale : BOOL ;
    tare_main_scale : BOOL ;
    cont_main_scale : BOOL ;
    zero_sub_scale : BOOL ;
    zero_cs : BOOL ;
    tare_cs : BOOL ;
    cont_cs : BOOL ;
    res64 : BOOL ;
    zero_lac_scale : BOOL ;
    tare_lac_scale : BOOL ;
    cont_lac_scale : BOOL ;
    Null_Abz2 : BOOL ;
    Tara_Abz2 : BOOL ;
    Inhalt_abz2 : BOOL ;
    res71 : BOOL ;
    res72 : BOOL ;
    filling_1 : BOOL ;
    filling_2 : BOOL ;
    filling_3 : BOOL ;
    filling_4 : BOOL ;
    filling_5 : BOOL ;
    filling_6 : BOOL ;
    filling_7 : BOOL ;
    filling_8 : BOOL ;
    fillvalve_1 : BOOL ;
    fillvalve_2 : BOOL ;
    fillvalve_3 : BOOL ;
    fillvalve_4 : BOOL ;
    fillvalve_5 : BOOL ;
    fillvalve_6 : BOOL ;
    fillvalve_7 : BOOL ;
    fillvalve_1_1 : BOOL ;
    fill_KK : ARRAY  [8 .. 17 ] OF BOOL  := FALSE;
    disc_ms_st1 : BOOL ;	//discharge main scale into storage vessel 1
    disc_ms_st2 : BOOL ;	//discharge main scale into storage vessel 2
    disc_ss : BOOL ;	//discharge sub scale
    res7 : ARRAY  [1 .. 1 ] OF WORD ;
   END_STRUCT ;
   Lamp : STRUCT
    main_start_G : BOOL ;
    stop_G : BOOL ;
    fault_G : BOOL ;
    horn_off : BOOL ;
    main_start_L : BOOL ;
    stop_L : BOOL ;
    fault_L : BOOL ;
    res84 : BOOL ;
    empty_W1 : BOOL ;
    empty_W2 : BOOL ;
    empty_W3 : BOOL ;
    empty_W4 : BOOL ;
    overload_W1 : BOOL ;
    overload_W2 : BOOL ;
    overload_W3 : BOOL ;
    overload_W4 : BOOL ;
    res : ARRAY  [1 .. 8 ] OF BYTE ;
    RW_HW : BYTE ;
    RW_V1 : BYTE ;
    RW_V2 : BYTE ;
    RW_V3 : BYTE ;
    RW_V4 : BYTE ;
    RW_V5 : BYTE ;
    RW_V6 : BYTE ;
    RW_V7 : BYTE ;
    RW_LW : BYTE ;
    Entl_HW_V1 : BYTE ;
    Entl_HW_V2 : BYTE ;
    Entl_HW_V3 : BYTE ;
    Entl_HW_V4 : BYTE ;
    Entl_HW_V5 : BYTE ;
    Entl_HW_V6 : BYTE ;
    Entl_LW_V1 : BYTE ;
    Entl_LW_V2 : BYTE ;
    Entl_SW : BYTE ;
    Entl_FW : BYTE ;
    Res22 : BYTE ;
    Res23 : BYTE ;
    Dosing : STRUCT
     C1 : BYTE ;
     C2 : BYTE ;
     C3 : BYTE ;
     C4 : BYTE ;
     C5 : BYTE ;
     C6_ms : BYTE ;
     C6_ss : BYTE ;
     C7 : BYTE ;
     C8 : BYTE ;
     C9 : BYTE ;
     C10 : BYTE ;
     C11 : BYTE ;
     C12 : BYTE ;
     C13 : BYTE ;
     C14 : BYTE ;
     C15 : BYTE ;
     C16 : BYTE ;
     C17 : BYTE ;
     C18 : BYTE ;
     C19 : BYTE ;
     C20 : BYTE ;
     C21 : BYTE ;
     C22 : BYTE ;
     C23 : BYTE ;
     C24 : BYTE ;
     C25 : BYTE ;
     C26 : BYTE ;
     C27 : BYTE ;
     C28 : BYTE ;
     C29 : BYTE ;
     C30 : BYTE ;
     C31 : BYTE ;
     C32 : BYTE ;
    END_STRUCT ;
    dosi_HW : BYTE ;
    dosi_SW : BYTE ;
    circulation_vessel1 : BYTE ;
    circulation_vessel2 : BYTE ;
    filling_1 : BYTE ;
    filling_2 : BYTE ;
    filling_3 : BYTE ;
    filling_4 : BYTE ;
    filling_5 : BYTE ;
    filling_6 : BYTE ;
    filling_7 : BYTE ;
    filling_8 : BYTE ;
    fill_valve1 : BYTE ;
    fill_valve2 : BYTE ;
    fill_valve3 : BYTE ;
    fill_valve4 : BYTE ;
    fill_valve5 : BYTE ;
    fill_valve6 : BYTE ;
    fill_valve7 : BYTE ;
    fill_valve1_1 : BYTE ;
    level_storage_1 : BYTE ;
    level_storage_2 : BYTE ;
    level_vat1 : BYTE ;
    level_storage_3 : BYTE ;
    level_coater : BYTE ;
    levelVITS6 : BYTE ;
    level_LW_storage1 : BYTE ;
    level_LW_storage2 : BYTE ;
    level_vat1_1 : BYTE ;
    schieber22_2 : BYTE ;
    schieber23_1 : BYTE ;
    schieber23_2 : BYTE ;
    circulation_HW_st2 : BYTE ;
    res7 : BYTE ;
    Start : ARRAY  [1 .. 8 ] OF BYTE ;
    Vorrat : ARRAY  [1 .. 8 ] OF STRUCT
     leer : BYTE ;
     abruf : BYTE ;
     voll : BYTE ;
    END_STRUCT ;
    fill_KK : ARRAY  [8 .. 17 ] OF BYTE ;
    level_KK : ARRAY  [8 .. 17 ] OF BYTE ;
   END_STRUCT ;
   LED : ARRAY  [1 .. 16 ] OF BOOL  := FALSE;
   Lamp_Heating : ARRAY  [1 .. 8 ] OF BYTE  := B#16#0;
  END_STRUCT ;	
BEGIN
   Button.auto_lacquer := TRUE;
   Button.fill_KK[8] := TRUE;
   Button.fill_KK[9] := TRUE;
   Button.fill_KK[10] := TRUE;
   Button.fill_KK[11] := TRUE;
   Button.fill_KK[12] := TRUE;
   Button.fill_KK[13] := TRUE;
   Button.fill_KK[14] := TRUE;
   Button.fill_KK[15] := TRUE;
   Button.fill_KK[16] := TRUE;
   Button.disc_ms_st1 := TRUE;
   Lamp.empty_W1 := TRUE;
   Lamp.empty_W2 := TRUE;
   Lamp.Entl_HW_V3 := B#16#2;
   Lamp.Entl_HW_V4 := B#16#2;
   Lamp.Entl_HW_V5 := B#16#2;
   Lamp.Dosing.C19 := B#16#2;
   Lamp.Dosing.C20 := B#16#2;
   Lamp.dosi_HW := B#16#2;
   Lamp.level_storage_1 := B#16#A;
   Lamp.level_storage_2 := B#16#A;
   Lamp.level_vat1 := B#16#A;
   Lamp.level_LW_storage1 := B#16#64;
   Lamp.level_LW_storage2 := B#16#64;
   Lamp.Vorrat[3].leer := B#16#1;
   Lamp.Vorrat[3].abruf := B#16#1;
   Lamp.Vorrat[6].voll := B#16#1;
   Lamp.Vorrat[7].abruf := B#16#1;
   Lamp.Vorrat[8].leer := B#16#1;
   Lamp.Vorrat[8].abruf := B#16#1;
   Lamp.level_KK[8] := B#16#4B;
   Lamp.level_KK[9] := B#16#4B;
   Lamp.level_KK[10] := B#16#4B;
   Lamp.level_KK[11] := B#16#4B;
   Lamp.level_KK[12] := B#16#4B;
   Lamp.level_KK[13] := B#16#4B;
   Lamp.level_KK[14] := B#16#64;
   Lamp.level_KK[15] := B#16#4B;
   Lamp.level_KK[16] := B#16#4B;
   Lamp.level_KK[17] := B#16#19;
END_DATA_BLOCK

DATA_BLOCK "SFC83_RETVAL_DB"	// DB 5
VERSION : 0.1
  STRUCT
   START1 : WORD ;
   START2 : WORD ;
   START3 : WORD ;
   START4 : WORD ;
   START5 : WORD ;
   START6 : WORD ;
   START7 : WORD ;
   START8 : WORD ;
  END_STRUCT ;	
BEGIN
   START4 := W#16#7000;
END_DATA_BLOCK

DATA_BLOCK "WScale1"	// DB 10
AUTHOR : Michel
VERSION : 0.0
"SiwarexCS"
BEGIN
END_DATA_BLOCK

DATA_BLOCK "WScale2"	// DB 11
AUTHOR : Michel
VERSION : 0.0
"SiwarexCS"
BEGIN
END_DATA_BLOCK

DATA_BLOCK "hornoff_DB"	// DB 19
VERSION : 0.0
  STRUCT
   Auftrag : STRUCT
    Nr : INT ;
    Par1 : INT ;
    Par2 : INT ;
    Par3 : INT ;
   END_STRUCT ;
   Datas : STRUCT
    RecipeNr : INT ;
    DataRecordNr : INT ;
    reseved1 : INT ;
    Status : STRUCT
     notused1 : BOOL ;
     notused2 : BOOL ;
     notused3 : BOOL ;
     notused4 : BOOL ;
     notused5 : BOOL ;
     notused6 : BOOL ;
     notused7 : BOOL ;
     notused8 : BOOL ;
     free : BOOL ;
     busy : BOOL ;
     ready : BOOL ;
     error : BOOL ;
    END_STRUCT ;
    reserved2 : INT ;
   END_STRUCT ;
   datetime : STRUCT
    year : BYTE ;
    month : BYTE ;
    day : BYTE ;
    hour : BYTE ;
    minute : BYTE ;
    second : BYTE ;
    res1 : BYTE ;
    weekday : BYTE ;	//low nibble!
    res2 : BYTE ;
    res3 : BYTE ;
    res4 : BYTE ;
    res5 : BYTE ;
   END_STRUCT ;
   LED : STRUCT
    OP1 : BOOL ;
    OP2 : BOOL ;
    OD1 : BOOL ;
    OD2 : BOOL ;
    V1 : BOOL ;
    V2 : BOOL ;
    R1 : BOOL ;
    R2 : BOOL ;
    BR1 : BOOL ;
    Br2 : BOOL ;
    C1 : BOOL ;
    C2 : BOOL ;
    Sys1 : BOOL ;
    Sys2 : BOOL ;
    SP1 : BOOL ;
    SP2 : BOOL ;
   END_STRUCT ;
   Picture : STRUCT
    p_type : INT ;
    p_nr : INT ;
    res1 : INT ;
    res2 : INT ;
    res3 : INT ;
   END_STRUCT ;
   reserve : ARRAY  [1 .. 15 ] OF WORD ;
   error_gravimet : ARRAY  [1 .. 160 ] OF
   BOOL ;
   quit_error_gravimet : ARRAY  [1 .. 160 ] OF
   BOOL ;
   error_ARP : ARRAY  [161 .. 320 ] OF BOOL ;
   quit_error_ARP : ARRAY  [161 .. 320 ] OF BOOL ;
  END_STRUCT ;	
BEGIN
END_DATA_BLOCK

DATA_BLOCK "HMI_Interf"	// DB 20
VERSION : 0.0
  STRUCT
   Auftrag : STRUCT
    Nr : INT ;
    Par1 : INT ;
    Par2 : INT ;
    Par3 : INT ;
   END_STRUCT ;
   Datas : STRUCT
    RecipeNr : INT ;
    DataRecordNr : INT ;
    reseved1 : INT ;
    Status : STRUCT
     notused1 : BOOL ;
     notused2 : BOOL ;
     notused3 : BOOL ;
     notused4 : BOOL ;
     notused5 : BOOL ;
     notused6 : BOOL ;
     notused7 : BOOL ;
     notused8 : BOOL ;
     free : BOOL ;
     busy : BOOL ;
     ready : BOOL ;
     error : BOOL ;
    END_STRUCT ;
    reserved2 : INT ;
    date_time : STRUCT
     dt_OP : DATE_AND_TIME ;
     res1 : BYTE ;
     res2 : BYTE ;
     res3 : BYTE ;
     res4 : BYTE ;
    END_STRUCT ;
   END_STRUCT ;
   LED : STRUCT
    OP1 : BOOL ;
    OP2 : BOOL ;
    OD1 : BOOL ;
    OD2 : BOOL ;
    V1 : BOOL ;
    V2 : BOOL ;
    R1 : BOOL ;
    R2 : BOOL ;
    BR1 : BOOL ;
    Br2 : BOOL ;
    C1 : BOOL ;
    C2 : BOOL ;
    Sys1 : BOOL ;
    Sys2 : BOOL ;
    SP1 : BOOL ;
    SP2 : BOOL ;
   END_STRUCT ;
   Picture : STRUCT
    p_type : INT ;
    p_nr : INT ;
    res1 : INT ;
    res2 : INT ;
    res3 : INT ;
   END_STRUCT ;
   reserve : ARRAY  [1 .. 15 ] OF WORD ;
   error : ARRAY  [1 .. 30 ] OF WORD ;
   quit_error : ARRAY  [1 .. 30 ] OF WORD ;
  END_STRUCT ;	
BEGIN
   Datas.RecipeNr := 1;
   Datas.DataRecordNr := 199;
   LED.OP1 := TRUE;
   LED.OP2 := TRUE;
   Picture.p_type := 1;
   Picture.p_nr := 12;
   Picture.res2 := 14;
   reserve[2] := W#16#5;
   reserve[5] := W#16#A2;
   reserve[6] := W#16#A1;
   quit_error[11] := W#16#800;
END_DATA_BLOCK

DATA_BLOCK "Auto_DB"	// DB 21
VERSION : 0.0
  STRUCT
   Step_scale1 : INT ;
   Step_scale2 : INT ;
   Step_scale3 : INT ;
   Start_G : BYTE ;
   rem_start1L : BOOL ;
   rem_start2L : BOOL ;
   reserve1 : BOOL ;
   reserve2 : BOOL ;
   reserve3 : BOOL ;
   reserve4 : BOOL ;
   reserve5 : BOOL ;
   reserve6 : BOOL ;
   rem_start1 : BOOL ;
   rem_start2 : BOOL ;
   rem_start3 : BOOL ;
   rem_start4 : BOOL ;
   rem_start5 : BOOL ;
   rem_start6 : BOOL ;
   rem_start7 : BOOL ;
   rem_start8 : BOOL ;
   automatic : BOOL ;
   automatic_L : BOOL ;
   Step_scale5 : INT ;
   Start_L : BYTE ;
  END_STRUCT ;	
BEGIN
   Step_scale1 := 24;
   Step_scale2 := 24;
   Step_scale3 := 24;
   Start_G := B#16#1;
   Start_L := B#16#2;
END_DATA_BLOCK

DATA_BLOCK "RecDB"	// DB 22
VERSION : 0.1
  STRUCT
   step : ARRAY  [1 .. 25 ] OF UDT 1;
   step_res : ARRAY  [26 .. 35 ] OF UDT 1;
   rec_save : BOOL ;
   rec_delete : BOOL ;
   PC1_active : BOOL ;
   MP1_active : BOOL ;
   res : BOOL ;
   res1 : BOOL ;
   res2 : BOOL ;
   res3 : BOOL ;
   rec_copy : BOOL ;
   rec_cut : BOOL ;
   rec_paste : BOOL ;
   rec_new : INT ;
   rec_old : INT ;
   compare_recipe : BOOL ;
   overwrite_recipe : BOOL ;
   no_overwrite_recipe : BOOL ;
   busy_trans : BOOL ;
   busy_save : BOOL ;
  END_STRUCT ;	
BEGIN
   step[1].Action := 769;
   step[1].comp := 17;
   step[1].rated_val := 2.000000e+00;
   rec_new := 77;
   rec_old := 77;
END_DATA_BLOCK

DATA_BLOCK "HMI_DB"	// DB 23
VERSION : 0.1
  STRUCT
   printerr : BOOL ;
   clear_cons : BOOL ;
   clear_OP : BOOL ;
   print_BR : BOOL ;
   fetch_clk : BOOL ;
   disc_sub : BOOL ;
   del_line : BOOL ;
   ins_line : BOOL ;
   screw : BOOL ;
   pump : BOOL ;
   print_BR_L : BOOL ;
   fill_vat : BOOL ;
   fill_coater : BOOL ;
   fill_ARP_coating : BOOL ;
   ARP_coating : BOOL ;
   disc_P : BOOL ;
   level : ARRAY  [1 .. 8 ] OF BYTE ;
   blk_ret_val : INT ;
   rez_line : INT ;
   disc_main : BYTE ;
   disc_col : BYTE ;
   Scale1_timers : STRUCT
    sec : INT ;
    min : INT ;
   END_STRUCT ;
   Scale2_timers : STRUCT
    sec : INT ;
    min : INT ;
   END_STRUCT ;
   Scale3_timers : STRUCT
    sec : INT ;
    min : INT ;
   END_STRUCT ;
   Scale4_timers : STRUCT
    sec : INT ;
    min : INT ;
   END_STRUCT ;
   BR_DB : INT  := 24;
   CP_DB_WRITE : INT ;
   CP_DB_READ : INT ;
   CP_DB_WRITE_P : INT ;
   CP_DB_READ_P : INT ;
   DelLine : INT ;
   db_BR_print : INT  := 124;
   print : BYTE ;	//0=no print // 1=print by fault // 2=print continuous
  END_STRUCT ;	
BEGIN
   printerr := TRUE;
   level[1] := B#16#2;
   level[2] := B#16#2;
   level[3] := B#16#2;
   level[4] := B#16#F;
   level[5] := B#16#2;
   level[6] := B#16#2;
   level[7] := B#16#64;
   level[8] := B#16#64;
   disc_main := B#16#10;
   BR_DB := 166;
   CP_DB_WRITE := 160;
   CP_DB_READ := 160;
   CP_DB_WRITE_P := 173;
   CP_DB_READ_P := 172;
   db_BR_print := 124;
END_DATA_BLOCK

DATA_BLOCK "BR_DB"	// DB 24
VERSION : 0.0
  STRUCT
   Recipe : INT ;
   batches : DINT ;
   Start : INT ;
   batchtime : DATE_AND_TIME ;
   header : ARRAY  [1 .. 7 ] OF INT ;
   BR : ARRAY  [1 .. 25 ] OF UDT 3;
  END_STRUCT ;	
BEGIN
   Recipe := 4;
   batches := L#52;
   Start := 1;
   BR[1].comp_nr := 1;
   BR[1].rated_val := 1.750000e+02;
   BR[1].real_val := 1.747850e+02;
   BR[2].comp_nr := 2;
   BR[2].rated_val := 7.500000e+01;
   BR[2].real_val := 7.492393e+01;
   BR[3].comp_nr := 8;
   BR[3].rated_val := 6.000000e-01;
   BR[3].real_val := 6.006358e-01;
   BR[4].comp_nr := 10;
   BR[4].rated_val := 1.480000e+00;
   BR[4].real_val := 1.509955e+00;
   BR[5].comp_nr := 12;
   BR[5].rated_val := 1.000000e+00;
   BR[5].real_val := 1.001338e+00;
   BR[6].comp_nr := 6;
   BR[6].rated_val := 1.500000e+01;
   BR[6].real_val := 1.503430e+01;
   BR[7].comp_nr := 7;
   BR[7].rated_val := 1.600000e+00;
   BR[7].real_val := 1.597957e+00;
   BR[8].comp_nr := 7;
   BR[8].rated_val := 1.500000e+00;
   BR[8].real_val := 1.519185e+00;
END_DATA_BLOCK

DATA_BLOCK "Start_DB"	// DB 25
VERSION : 0.0
  STRUCT
   Start : ARRAY  [1 .. 8 ] OF UDT 2;
  END_STRUCT ;	
BEGIN
   Start[1].Prozent := 100;
   Start[2].Prozent := 100;
   Start[3].Prozent := 100;
   Start[4].Prozent := 100;
   Start[5].Prozent := 100;
   Start[6].Prozent := 100;
   Start[7].Prozent := 100;
   Start[8].Prozent := 100;
END_DATA_BLOCK

DATA_BLOCK "WorkDB-G"	// DB 26
VERSION : 0.0
  STRUCT
   step : ARRAY  [1 .. 25 ] OF UDT 1;
  END_STRUCT ;	
BEGIN
   step[1].Action := 257;
   step[1].comp := 2;
   step[1].rated_val := 2.000000e+00;
   step[2].Action := 257;
   step[2].comp := 3;
   step[2].rated_val := 2.000000e+00;
   step[3].Action := 515;
   step[3].comp := 6;
   step[3].rated_val := 2.000000e-01;
   step[4].Action := 515;
   step[4].comp := 7;
   step[4].rated_val := 2.000000e-01;
   step[5].Action := 515;
   step[5].comp := 8;
   step[5].rated_val := 2.000000e-01;
   step[6].Action := 515;
   step[6].comp := 9;
   step[6].rated_val := 2.000000e-01;
   step[7].Action := 515;
   step[7].comp := 10;
   step[7].rated_val := 2.000000e-01;
   step[8].Action := 515;
   step[8].comp := 11;
   step[8].agit_time := 40;
   step[8].rated_val := 2.000000e-01;
   step[9].Action := 259;
   step[9].comp := 11;
   step[9].rated_val := 1.401298e-45;
   step[10].Action := 257;
   step[10].comp := 5;
   step[10].rated_val := 5.000000e+00;
   step[11].Action := 259;
   step[11].comp := 5;
   step[11].rated_val := 1.401298e-45;
END_DATA_BLOCK

DATA_BLOCK "speed_DB"	// DB 27
VERSION : 0.0
  STRUCT
   act_val : INT  := 1250;	//range 0..2500
   dosing_high : INT  := 2500;	//range 0..2500
   Temp_V1 : INT ;	//Temperatur des Vorratsbehälter 1
   Temp_V2 : INT ;	//Temperatur des Vorratsbehälter 2
   reserve : ARRAY  [1 .. 12 ] OF INT ;
   mixtime : ARRAY  [1 .. 8 ] OF //auto mix time while discharging
   S5TIME  := S5T#1M;
  END_STRUCT ;	
BEGIN
   dosing_high := 2500;
   Temp_V1 := 308;
   Temp_V2 := 304;
   mixtime[1] := S5T#2M;
   mixtime[2] := S5T#2M;
   mixtime[3] := S5T#1M;
   mixtime[4] := S5T#1M;
   mixtime[5] := S5T#1M;
   mixtime[6] := S5T#1M;
   mixtime[7] := S5T#1M;
   mixtime[8] := S5T#1M;
END_DATA_BLOCK

DATA_BLOCK "comp0"	// DB 30
VERSION : 0.0
  STRUCT
   tank : REAL ;
   verbrauch : REAL ;
   grobfein : REAL ;
   toleranz : REAL ;
   nachlauf : REAL ;
   ruehrzeit : INT ;
   kompname : STRING  [16 ];
   fuellung : REAL ;
  END_STRUCT ;	
BEGIN
END_DATA_BLOCK

DATA_BLOCK "comp1"	// DB 31
VERSION : 0.0
  STRUCT
   tank : REAL ;
   verbrauch : REAL ;
   grobfein : REAL ;
   toleranz : REAL ;
   nachlauf : REAL ;
   ruehrzeit : INT ;
   kompname : STRING  [16 ];
   fuellung : REAL ;
  END_STRUCT ;	
BEGIN
END_DATA_BLOCK

DATA_BLOCK "comp2"	// DB 32
VERSION : 0.0
  STRUCT
   tank : REAL ;
   verbrauch : REAL ;
   grobfein : REAL ;
   toleranz : REAL ;
   nachlauf : REAL ;
   ruehrzeit : INT ;
   kompname : STRING  [16 ];
   fuellung : REAL ;
  END_STRUCT ;	
BEGIN
END_DATA_BLOCK

DATA_BLOCK "comp3"	// DB 33
VERSION : 0.0
  STRUCT
   tank : REAL ;
   verbrauch : REAL ;
   grobfein : REAL ;
   toleranz : REAL ;
   nachlauf : REAL ;
   ruehrzeit : INT ;
   kompname : STRING  [16 ];
   fuellung : REAL ;
  END_STRUCT ;	
BEGIN
END_DATA_BLOCK

DATA_BLOCK "comp4"	// DB 34
VERSION : 0.0
  STRUCT
   tank : REAL ;
   verbrauch : REAL ;
   grobfein : REAL ;
   toleranz : REAL ;
   nachlauf : REAL ;
   ruehrzeit : INT ;
   kompname : STRING  [16 ];
   fuellung : REAL ;
  END_STRUCT ;	
BEGIN
END_DATA_BLOCK

DATA_BLOCK "comp5"	// DB 35
VERSION : 0.0
  STRUCT
   tank : REAL ;
   verbrauch : REAL ;
   grobfein : REAL ;
   toleranz : REAL ;
   nachlauf : REAL ;
   ruehrzeit : INT ;
   kompname : STRING  [16 ];
   fuellung : REAL ;
  END_STRUCT ;	
BEGIN
END_DATA_BLOCK

DATA_BLOCK "comp6"	// DB 36
VERSION : 0.0
  STRUCT
   tank : REAL ;
   verbrauch : REAL ;
   grobfein : REAL ;
   toleranz : REAL ;
   nachlauf : REAL ;
   ruehrzeit : INT ;
   kompname : STRING  [16 ];
   fuellung : REAL ;
  END_STRUCT ;	
BEGIN
END_DATA_BLOCK

DATA_BLOCK "comp7"	// DB 37
VERSION : 0.0
  STRUCT
   tank : REAL ;
   verbrauch : REAL ;
   grobfein : REAL ;
   toleranz : REAL ;
   nachlauf : REAL ;
   ruehrzeit : INT ;
   kompname : STRING  [16 ];
   fuellung : REAL ;
  END_STRUCT ;	
BEGIN
END_DATA_BLOCK

DATA_BLOCK "comp8"	// DB 38
VERSION : 0.0
  STRUCT
   tank : REAL ;
   verbrauch : REAL ;
   grobfein : REAL ;
   toleranz : REAL ;
   nachlauf : REAL ;
   ruehrzeit : INT ;
   kompname : STRING  [16 ];
   fuellung : REAL ;
  END_STRUCT ;	
BEGIN
END_DATA_BLOCK

DATA_BLOCK "comp9"	// DB 39
VERSION : 0.0
  STRUCT
   tank : REAL ;
   verbrauch : REAL ;
   grobfein : REAL ;
   toleranz : REAL ;
   nachlauf : REAL ;
   ruehrzeit : INT ;
   kompname : STRING  [16 ];
   fuellung : REAL ;
  END_STRUCT ;	
BEGIN
END_DATA_BLOCK

DATA_BLOCK "comp10"	// DB 40
VERSION : 0.0
  STRUCT
   tank : REAL ;
   verbrauch : REAL ;
   grobfein : REAL ;
   toleranz : REAL ;
   nachlauf : REAL ;
   ruehrzeit : INT ;
   kompname : STRING  [16 ];
   fuellung : REAL ;
  END_STRUCT ;	
BEGIN
END_DATA_BLOCK

DATA_BLOCK "comp11"	// DB 41
VERSION : 0.0
  STRUCT
   tank : REAL ;
   verbrauch : REAL ;
   grobfein : REAL ;
   toleranz : REAL ;
   nachlauf : REAL ;
   ruehrzeit : INT ;
   kompname : STRING  [16 ];
   fuellung : REAL ;
  END_STRUCT ;	
BEGIN
END_DATA_BLOCK

DATA_BLOCK "comp12"	// DB 42
VERSION : 0.0
  STRUCT
   tank : REAL ;
   verbrauch : REAL ;
   grobfein : REAL ;
   toleranz : REAL ;
   nachlauf : REAL ;
   ruehrzeit : INT ;
   kompname : STRING  [16 ];
   fuellung : REAL ;
  END_STRUCT ;	
BEGIN
END_DATA_BLOCK

DATA_BLOCK "comp13"	// DB 43
VERSION : 0.0
  STRUCT
   tank : REAL ;
   verbrauch : REAL ;
   grobfein : REAL ;
   toleranz : REAL ;
   nachlauf : REAL ;
   ruehrzeit : INT ;
   kompname : STRING  [16 ];
   fuellung : REAL ;
  END_STRUCT ;	
BEGIN
END_DATA_BLOCK

DATA_BLOCK "comp14"	// DB 44
VERSION : 0.0
  STRUCT
   tank : REAL ;
   verbrauch : REAL ;
   grobfein : REAL ;
   toleranz : REAL ;
   nachlauf : REAL ;
   ruehrzeit : INT ;
   kompname : STRING  [16 ];
   fuellung : REAL ;
  END_STRUCT ;	
BEGIN
END_DATA_BLOCK

DATA_BLOCK "comp15"	// DB 45
VERSION : 0.0
  STRUCT
   tank : REAL ;
   verbrauch : REAL ;
   grobfein : REAL ;
   toleranz : REAL ;
   nachlauf : REAL ;
   ruehrzeit : INT ;
   kompname : STRING  [16 ];
   fuellung : REAL ;
  END_STRUCT ;	
BEGIN
END_DATA_BLOCK

DATA_BLOCK "comp16"	// DB 46
VERSION : 0.0
  STRUCT
   tank : REAL ;
   verbrauch : REAL ;
   grobfein : REAL ;
   toleranz : REAL ;
   nachlauf : REAL ;
   ruehrzeit : INT ;
   kompname : STRING  [16 ];
   fuellung : REAL ;
  END_STRUCT ;	
BEGIN
END_DATA_BLOCK

DATA_BLOCK "comp17"	// DB 47
VERSION : 0.0
  STRUCT
   tank : REAL ;
   verbrauch : REAL ;
   grobfein : REAL ;
   toleranz : REAL ;
   nachlauf : REAL ;
   ruehrzeit : INT ;
   kompname : STRING  [16 ];
   fuellung : REAL ;
  END_STRUCT ;	
BEGIN
END_DATA_BLOCK

DATA_BLOCK "comp18"	// DB 48
VERSION : 0.0
  STRUCT
   tank : REAL ;
   verbrauch : REAL ;
   grobfein : REAL ;
   toleranz : REAL ;
   nachlauf : REAL ;
   ruehrzeit : INT ;
   kompname : STRING  [16 ];
   fuellung : REAL ;
  END_STRUCT ;	
BEGIN
END_DATA_BLOCK

DATA_BLOCK "comp19"	// DB 49
VERSION : 0.0
  STRUCT
   tank : REAL ;
   verbrauch : REAL ;
   grobfein : REAL ;
   toleranz : REAL ;
   nachlauf : REAL ;
   ruehrzeit : INT ;
   kompname : STRING  [16 ];
   fuellung : REAL ;
  END_STRUCT ;	
BEGIN
END_DATA_BLOCK

DATA_BLOCK "comp20"	// DB 50
VERSION : 0.0
  STRUCT
   tank : REAL ;
   verbrauch : REAL ;
   grobfein : REAL ;
   toleranz : REAL ;
   nachlauf : REAL ;
   ruehrzeit : INT ;
   kompname : STRING  [16 ];
   fuellung : REAL ;
  END_STRUCT ;	
BEGIN
END_DATA_BLOCK

DATA_BLOCK "comp21"	// DB 51
VERSION : 0.0
  STRUCT
   tank : REAL ;
   verbrauch : REAL ;
   grobfein : REAL ;
   toleranz : REAL ;
   nachlauf : REAL ;
   ruehrzeit : INT ;
   kompname : STRING  [16 ];
   fuellung : REAL ;
  END_STRUCT ;	
BEGIN
END_DATA_BLOCK

DATA_BLOCK "comp22"	// DB 52
VERSION : 0.0
  STRUCT
   tank : REAL ;
   verbrauch : REAL ;
   grobfein : REAL ;
   toleranz : REAL ;
   nachlauf : REAL ;
   ruehrzeit : INT ;
   kompname : STRING  [16 ];
   fuellung : REAL ;
  END_STRUCT ;	
BEGIN
END_DATA_BLOCK

DATA_BLOCK "comp23"	// DB 53
VERSION : 0.0
  STRUCT
   tank : REAL ;
   verbrauch : REAL ;
   grobfein : REAL ;
   toleranz : REAL ;
   nachlauf : REAL ;
   ruehrzeit : INT ;
   kompname : STRING  [16 ];
   fuellung : REAL ;
  END_STRUCT ;	
BEGIN
END_DATA_BLOCK

DATA_BLOCK "comp24"	// DB 54
VERSION : 0.0
  STRUCT
   tank : REAL ;
   verbrauch : REAL ;
   grobfein : REAL ;
   toleranz : REAL ;
   nachlauf : REAL ;
   ruehrzeit : INT ;
   kompname : STRING  [16 ];
   fuellung : REAL ;
  END_STRUCT ;	
BEGIN
END_DATA_BLOCK

DATA_BLOCK "comp25"	// DB 55
VERSION : 0.0
  STRUCT
   tank : REAL ;
   verbrauch : REAL ;
   grobfein : REAL ;
   toleranz : REAL ;
   nachlauf : REAL ;
   ruehrzeit : INT ;
   kompname : STRING  [16 ];
   fuellung : REAL ;
  END_STRUCT ;	
BEGIN
END_DATA_BLOCK

DATA_BLOCK "comp26"	// DB 56
VERSION : 0.0
  STRUCT
   tank : REAL ;
   verbrauch : REAL ;
   grobfein : REAL ;
   toleranz : REAL ;
   nachlauf : REAL ;
   ruehrzeit : INT ;
   kompname : STRING  [16 ];
   fuellung : REAL ;
  END_STRUCT ;	
BEGIN
END_DATA_BLOCK

DATA_BLOCK "comp27"	// DB 57
VERSION : 0.0
  STRUCT
   tank : REAL ;
   verbrauch : REAL ;
   grobfein : REAL ;
   toleranz : REAL ;
   nachlauf : REAL ;
   ruehrzeit : INT ;
   kompname : STRING  [16 ];
   fuellung : REAL ;
  END_STRUCT ;	
BEGIN
END_DATA_BLOCK

DATA_BLOCK "comp28"	// DB 58
VERSION : 0.0
  STRUCT
   tank : REAL ;
   verbrauch : REAL ;
   grobfein : REAL ;
   toleranz : REAL ;
   nachlauf : REAL ;
   ruehrzeit : INT ;
   kompname : STRING  [16 ];
   fuellung : REAL ;
  END_STRUCT ;	
BEGIN
END_DATA_BLOCK

DATA_BLOCK "comp29"	// DB 59
VERSION : 0.0
  STRUCT
   tank : REAL ;
   verbrauch : REAL ;
   grobfein : REAL ;
   toleranz : REAL ;
   nachlauf : REAL ;
   ruehrzeit : INT ;
   kompname : STRING  [16 ];
   fuellung : REAL ;
  END_STRUCT ;	
BEGIN
END_DATA_BLOCK

DATA_BLOCK "comp30"	// DB 60
VERSION : 0.0
  STRUCT
   tank : REAL ;
   verbrauch : REAL ;
   grobfein : REAL ;
   toleranz : REAL ;
   nachlauf : REAL ;
   ruehrzeit : INT ;
   kompname : STRING  [16 ];
   fuellung : REAL ;
  END_STRUCT ;	
BEGIN
END_DATA_BLOCK

DATA_BLOCK "StartSeriesDB"	// DB 90
VERSION : 0.0
  STRUCT
   buffer : ARRAY  [1 .. 10 ] OF BYTE ;
   ptr : DINT ;
   FP : BYTE ;
  END_STRUCT ;	
BEGIN
END_DATA_BLOCK

DATA_BLOCK "DScale1"	// DB 100
VERSION : 0.0
"Dosing"
BEGIN
END_DATA_BLOCK

DATA_BLOCK "DScale2"	// DB 101
VERSION : 0.0
"Dosing"
BEGIN
END_DATA_BLOCK

DATA_BLOCK "DScale3"	// DB 102
VERSION : 0.0
"Dosing"
BEGIN
END_DATA_BLOCK

DATA_BLOCK "Rec_copy_DB"	// DB 122
TITLE = Data block for copying recipes(buffer)
VERSION : 0.1
  STRUCT
   step : ARRAY  [1 .. 25 ] OF UDT 1;
   step_res : ARRAY  [26 .. 35 ] OF UDT 1;
  END_STRUCT ;	
BEGIN
   step[1].Action := 257;
   step[1].comp := 2;
   step[1].rated_val := 1.300000e+02;
   step[2].Action := 257;
   step[2].comp := 4;
   step[2].rated_val := 1.320000e+01;
   step[3].Action := 512;
   step[3].comp := 11;
   step[3].rated_val := 3.900000e-01;
   step[4].Action := 512;
   step[4].comp := 9;
   step[4].rated_val := 6.500000e-01;
   step[5].Action := 512;
   step[5].comp := 8;
   step[5].rated_val := 3.250000e-01;
   step[6].Action := 512;
   step[6].comp := 7;
   step[6].agit_time := 40;
   step[6].rated_val := 3.900000e-01;
   step[7].Action := 259;
   step[8].Action := 257;
   step[8].comp := 5;
   step[8].rated_val := 5.000000e+00;
   step[9].Action := 259;
END_DATA_BLOCK

DATA_BLOCK "compare_Rec_DB"	// DB 123
TITLE = Data block for copying recipes(buffer)
VERSION : 0.1
  STRUCT
   step : ARRAY  [1 .. 25 ] OF UDT 1;
   step_res : ARRAY  [26 .. 35 ] OF UDT 1;
  END_STRUCT ;	
BEGIN
   step[1].Action := 769;
   step[1].comp := 17;
   step[1].rated_val := 2.000000e+00;
END_DATA_BLOCK

DATA_BLOCK "PrintBR_DB"	// DB 124
VERSION : 0.1
  STRUCT
   Recipe : INT ;
   batches : DINT ;
   Start : INT ;
   batchtime : DATE_AND_TIME ;
   header : ARRAY  [1 .. 7 ] OF INT ;
   BR : ARRAY  [1 .. 25 ] OF UDT 3;
   Order : STRING  [20 ];
  END_STRUCT ;	
BEGIN
   Recipe := 199;
   batches := L#3;
   Start := 2;
   BR[1].comp_nr := 2;
   BR[1].rated_val := 2.000000e+00;
   BR[1].real_val := 2.111425e+00;
   BR[2].comp_nr := 4;
   BR[2].rated_val := 2.000000e+00;
   BR[2].real_val := 1.886806e+00;
   BR[3].comp_nr := 6;
   BR[3].rated_val := 2.000000e-01;
   BR[3].real_val := 1.992425e-01;
   BR[4].comp_nr := 7;
   BR[4].rated_val := 2.000000e-01;
   BR[4].real_val := 2.404084e-01;
   BR[5].comp_nr := 8;
   BR[5].rated_val := 2.000000e-01;
   BR[5].real_val := 2.066524e-01;
   BR[6].comp_nr := 9;
   BR[6].rated_val := 2.000000e-01;
   BR[6].real_val := 2.017125e-01;
   BR[7].comp_nr := 10;
   BR[7].rated_val := 2.000000e-01;
   BR[7].real_val := 2.074757e-01;
   BR[8].comp_nr := 11;
   BR[8].rated_val := 2.000000e-01;
   BR[8].real_val := 1.992426e-01;
   BR[10].comp_nr := 5;
   BR[10].rated_val := 5.000000e+00;
   BR[10].real_val := 4.975327e+00;
   Order := 'u5009587';
END_DATA_BLOCK

DATA_BLOCK "Rec_Start1"	// DB 150
VERSION : 0.1
  STRUCT
   step : ARRAY  [1 .. 25 ] OF UDT 1;
  END_STRUCT ;	
BEGIN
   step[1].Action := 257;
   step[1].comp := 2;
   step[1].rated_val := 1.300000e+02;
   step[2].Action := 257;
   step[2].comp := 4;
   step[2].rated_val := 1.320000e+01;
   step[3].Action := 512;
   step[3].comp := 11;
   step[3].rated_val := 3.900000e-01;
   step[4].Action := 512;
   step[4].comp := 9;
   step[4].rated_val := 6.500000e-01;
   step[5].Action := 512;
   step[5].comp := 8;
   step[5].rated_val := 3.250000e-01;
   step[6].Action := 512;
   step[6].comp := 7;
   step[6].agit_time := 40;
   step[6].rated_val := 3.900000e-01;
   step[7].Action := 259;
   step[8].Action := 257;
   step[8].comp := 5;
   step[8].rated_val := 5.000000e+00;
   step[9].Action := 259;
END_DATA_BLOCK

DATA_BLOCK "Rec_Start2"	// DB 151
VERSION : 0.1
  STRUCT
   step : ARRAY  [1 .. 25 ] OF UDT 1;
  END_STRUCT ;	
BEGIN
   step[1].Action := 257;
   step[1].comp := 1;
   step[1].rated_val := 1.270000e+02;
   step[2].Action := 257;
   step[2].comp := 4;
   step[2].rated_val := 1.660000e+01;
   step[3].Action := 512;
   step[3].comp := 11;
   step[3].rated_val := 3.800000e-01;
   step[4].Action := 512;
   step[4].comp := 9;
   step[4].rated_val := 6.350000e-01;
   step[5].Action := 512;
   step[5].comp := 8;
   step[5].rated_val := 3.200000e-01;
   step[6].Action := 512;
   step[6].comp := 6;
   step[6].agit_time := 40;
   step[6].rated_val := 3.800000e-01;
   step[7].Action := 259;
   step[8].Action := 257;
   step[8].comp := 5;
   step[8].rated_val := 5.000000e+00;
   step[9].Action := 259;
END_DATA_BLOCK

DATA_BLOCK "Rec_Start3"	// DB 152
VERSION : 0.1
  STRUCT
   step : ARRAY  [1 .. 25 ] OF UDT 1;
  END_STRUCT ;	
BEGIN
   step[1].Action := 769;
   step[1].comp := 17;
   step[1].rated_val := 2.000000e+00;
END_DATA_BLOCK

